   1:L PR[91] 10mm/sec FINE;
   1:  PR[GP1:91,1] = PR[GP1:90,1] + 127.618;
   1:  PR[GP1:91,2] = PR[GP1:90,2] + 91.510;
   1:L PR[91] 10mm/sec FINE;
   1:  PR[GP1:91,1] = PR[GP1:90,1] + 127.930;
   1:  PR[GP1:91,2] = PR[GP1:90,2] + 92.754;
   1:L PR[91] 10mm/sec FINE;
   1:  PR[GP1:91,1] = PR[GP1:90,1] + 128.133;
   1:  PR[GP1:91,2] = PR[GP1:90,2] + 93.973;
   1:L PR[91] 10mm/sec FINE;
   1:  PR[GP1:91,1] = PR[GP1:90,1] + 128.288;
   1:  PR[GP1:91,2] = PR[GP1:90,2] + 95.442;
   1:L PR[91] 10mm/sec FINE;
   1:  PR[GP1:91,1] = PR[GP1:90,1] + 128.356;
   1:  PR[GP1:91,2] = PR[GP1:90,2] + 96.587;
   1:L PR[91] 10mm/sec FINE;
   1:  PR[GP1:91,1] = PR[GP1:90,1] + 128.349;
   1:  PR[GP1:91,2] = PR[GP1:90,2] + 97.306;
   1:L PR[91] 10mm/sec FINE;
   1:  PR[GP1:91,1] = PR[GP1:90,1] + 128.144;
   1:  PR[GP1:91,2] = PR[GP1:90,2] + 98.735;
   1:L PR[91] 10mm/sec FINE;
   1:  PR[GP1:91,1] = PR[GP1:90,1] + 127.993;
   1:  PR[GP1:91,2] = PR[GP1:90,2] + 100.189;
   1:L PR[91] 10mm/sec FINE;
   1:  PR[GP1:91,1] = PR[GP1:90,1] + 127.642;
   1:  PR[GP1:91,2] = PR[GP1:90,2] + 101.364;
   1:L PR[91] 10mm/sec FINE;
   1:  PR[GP1:91,1] = PR[GP1:90,1] + 126.916;
   1:  PR[GP1:91,2] = PR[GP1:90,2] + 104.069;
   1:L PR[91] 10mm/sec FINE;
   1:  PR[GP1:91,1] = PR[GP1:90,1] + 125.251;
   1:  PR[GP1:91,2] = PR[GP1:90,2] + 107.811;
   1:L PR[91] 10mm/sec FINE;
   1:  PR[GP1:91,1] = PR[GP1:90,1] + 122.955;
   1:  PR[GP1:91,2] = PR[GP1:90,2] + 111.333;
   1:L PR[91] 10mm/sec FINE;
   1:  PR[GP1:91,1] = PR[GP1:90,1] + 121.825;
   1:  PR[GP1:91,2] = PR[GP1:90,2] + 112.546;
   1:L PR[91] 10mm/sec FINE;
   1:  PR[GP1:91,1] = PR[GP1:90,1] + 120.143;
   1:  PR[GP1:91,2] = PR[GP1:90,2] + 114.425;
   1:L PR[91] 10mm/sec FINE;
   1:  PR[GP1:91,1] = PR[GP1:90,1] + 118.607;
   1:  PR[GP1:91,2] = PR[GP1:90,2] + 115.642;
   1:L PR[91] 10mm/sec FINE;
   1:  PR[GP1:91,1] = PR[GP1:90,1] + 116.943;
   1:  PR[GP1:91,2] = PR[GP1:90,2] + 116.933;
   1:L PR[91] 10mm/sec FINE;
   1:  PR[GP1:91,1] = PR[GP1:90,1] + 113.463;
   1:  PR[GP1:91,2] = PR[GP1:90,2] + 118.770;
   1:L PR[91] 10mm/sec FINE;
   1:  PR[GP1:91,1] = PR[GP1:90,1] + 109.869;
   1:  PR[GP1:91,2] = PR[GP1:90,2] + 119.883;
   1:L PR[91] 10mm/sec FINE;
   1:  PR[GP1:91,1] = PR[GP1:90,1] + 108.820;
   1:  PR[GP1:91,2] = PR[GP1:90,2] + 120.007;
   1:L PR[91] 10mm/sec FINE;
   1:  PR[GP1:91,1] = PR[GP1:90,1] + 106.260;
   1:  PR[GP1:91,2] = PR[GP1:90,2] + 120.260;
   1:L PR[91] 10mm/sec FINE;
   1:  PR[GP1:91,1] = PR[GP1:90,1] + 104.599;
   1:  PR[GP1:91,2] = PR[GP1:90,2] + 120.142;
   1:L PR[91] 10mm/sec FINE;
   1:  PR[GP1:91,1] = PR[GP1:90,1] + 102.606;
   1:  PR[GP1:91,2] = PR[GP1:90,2] + 119.945;
   1:L PR[91] 10mm/sec FINE;
   1:  PR[GP1:91,1] = PR[GP1:90,1] + 101.931;
   1:  PR[GP1:91,2] = PR[GP1:90,2] + 119.914;
   1:L PR[91] 10mm/sec FINE;
   1:  PR[GP1:91,1] = PR[GP1:90,1] + 98.093;
   1:  PR[GP1:91,2] = PR[GP1:90,2] + 119.921;
   1:L PR[91] 10mm/sec FINE;
   1:  PR[GP1:91,1] = PR[GP1:90,1] + 97.212;
   1:  PR[GP1:91,2] = PR[GP1:90,2] + 119.946;
   1:L PR[91] 10mm/sec FINE;
   1:  PR[GP1:91,1] = PR[GP1:90,1] + 94.419;
   1:  PR[GP1:91,2] = PR[GP1:90,2] + 119.458;
   1:L PR[91] 10mm/sec FINE;
   1:  PR[GP1:91,1] = PR[GP1:90,1] + 92.766;
   1:  PR[GP1:91,2] = PR[GP1:90,2] + 119.217;
   1:L PR[91] 10mm/sec FINE;
   1:  PR[GP1:91,1] = PR[GP1:90,1] + 90.935;
   1:  PR[GP1:91,2] = PR[GP1:90,2] + 118.517;
   1:L PR[91] 10mm/sec FINE;
   1:  PR[GP1:91,1] = PR[GP1:90,1] + 88.767;
   1:  PR[GP1:91,2] = PR[GP1:90,2] + 117.763;
   1:L PR[91] 10mm/sec FINE;
   1:  PR[GP1:91,1] = PR[GP1:90,1] + 87.721;
   1:  PR[GP1:91,2] = PR[GP1:90,2] + 117.075;
   1:L PR[91] 10mm/sec FINE;
   1:  PR[GP1:91,1] = PR[GP1:90,1] + 85.366;
   1:  PR[GP1:91,2] = PR[GP1:90,2] + 115.642;
   1:L PR[91] 10mm/sec FINE;
   1:  PR[GP1:91,1] = PR[GP1:90,1] + 84.875;
   1:  PR[GP1:91,2] = PR[GP1:90,2] + 115.109;
   1:L PR[91] 10mm/sec FINE;
   1:  PR[GP1:91,1] = PR[GP1:90,1] + 82.710;
   1:  PR[GP1:91,2] = PR[GP1:90,2] + 112.923;
   1:L PR[91] 10mm/sec FINE;
   1:  PR[GP1:91,1] = PR[GP1:90,1] + 82.531;
   1:  PR[GP1:91,2] = PR[GP1:90,2] + 112.581;
   1:L PR[91] 10mm/sec FINE;
   1:  PR[GP1:91,1] = PR[GP1:90,1] + 80.884;
   1:  PR[GP1:91,2] = PR[GP1:90,2] + 109.710;
   1:L PR[91] 10mm/sec FINE;
   1:  PR[GP1:91,1] = PR[GP1:90,1] + 80.830;
   1:  PR[GP1:91,2] = PR[GP1:90,2] + 109.475;
   1:L PR[91] 10mm/sec FINE;
   1:  PR[GP1:91,1] = PR[GP1:90,1] + 79.909;
   1:  PR[GP1:91,2] = PR[GP1:90,2] + 106.150;
   1:L PR[91] 10mm/sec FINE;
   1:  PR[GP1:91,1] = PR[GP1:90,1] + 79.999;
   1:  PR[GP1:91,2] = PR[GP1:90,2] + 102.825;
   1:L PR[91] 10mm/sec FINE;
   1:  PR[GP1:91,1] = PR[GP1:90,1] + 80.036;
   1:  PR[GP1:91,2] = PR[GP1:90,2] + 102.315;
   1:L PR[91] 10mm/sec FINE;
   1:  PR[GP1:91,1] = PR[GP1:90,1] + 80.087;
   1:  PR[GP1:91,2] = PR[GP1:90,2] + 102.069;
   1:L PR[91] 10mm/sec FINE;
   1:  PR[GP1:91,1] = PR[GP1:90,1] + 80.782;
   1:  PR[GP1:91,2] = PR[GP1:90,2] + 99.840;
   1:L PR[91] 10mm/sec FINE;
   1:  PR[GP1:91,1] = PR[GP1:90,1] + 81.137;
   1:  PR[GP1:91,2] = PR[GP1:90,2] + 98.649;
   1:L PR[91] 10mm/sec FINE;
   1:  PR[GP1:91,1] = PR[GP1:90,1] + 81.314;
   1:  PR[GP1:91,2] = PR[GP1:90,2] + 98.024;
   1:L PR[91] 10mm/sec FINE;
   1:  PR[GP1:91,1] = PR[GP1:90,1] + 81.395;
   1:  PR[GP1:91,2] = PR[GP1:90,2] + 97.791;
   1:L PR[91] 10mm/sec FINE;
   1:  PR[GP1:91,1] = PR[GP1:90,1] + 83.374;
   1:  PR[GP1:91,2] = PR[GP1:90,2] + 94.282;
   1:L PR[91] 10mm/sec FINE;
   1:  PR[GP1:91,1] = PR[GP1:90,1] + 84.843;
   1:  PR[GP1:91,2] = PR[GP1:90,2] + 92.903;
   1:  PR[GP1:91,3] = PR[GP1:90,3] + 54.900;
   1:L PR[91] 10mm/sec FINE;
   1:  PR[GP1:91,1] = PR[GP1:90,1] + 86.776;
   1:  PR[GP1:91,2] = PR[GP1:90,2] + 90.767;
   1:L PR[91] 10mm/sec FINE;
   1:  PR[GP1:91,1] = PR[GP1:90,1] + 88.811;
   1:  PR[GP1:91,2] = PR[GP1:90,2] + 88.734;
   1:L PR[91] 10mm/sec FINE;
   1:  PR[GP1:91,1] = PR[GP1:90,1] + 90.211;
   1:  PR[GP1:91,2] = PR[GP1:90,2] + 87.682;
   1:L PR[91] 10mm/sec FINE;
   1:  PR[GP1:91,1] = PR[GP1:90,1] + 93.880;
   1:  PR[GP1:91,2] = PR[GP1:90,2] + 85.209;
   1:L PR[91] 10mm/sec FINE;
   1:  PR[GP1:91,1] = PR[GP1:90,1] + 94.184;
   1:  PR[GP1:91,2] = PR[GP1:90,2] + 85.056;
   1:L PR[91] 10mm/sec FINE;
   1:  PR[GP1:91,1] = PR[GP1:90,1] + 95.228;
   1:  PR[GP1:91,2] = PR[GP1:90,2] + 84.601;
   1:L PR[91] 10mm/sec FINE;
   1:  PR[GP1:91,1] = PR[GP1:90,1] + 99.096;
   1:  PR[GP1:91,2] = PR[GP1:90,2] + 82.673;
   1:L PR[91] 10mm/sec FINE;
   1:  PR[GP1:91,1] = PR[GP1:90,1] + 100.630;
   1:  PR[GP1:91,2] = PR[GP1:90,2] + 82.156;
   1:L PR[91] 10mm/sec FINE;
   1:  PR[GP1:91,1] = PR[GP1:90,1] + 104.317;
   1:  PR[GP1:91,2] = PR[GP1:90,2] + 81.077;
   1:L PR[91] 10mm/sec FINE;
   1:  PR[GP1:91,1] = PR[GP1:90,1] + 107.737;
   1:  PR[GP1:91,2] = PR[GP1:90,2] + 80.558;
   1:L PR[91] 10mm/sec FINE;
   1:  PR[GP1:91,1] = PR[GP1:90,1] + 109.469;
   1:  PR[GP1:91,2] = PR[GP1:90,2] + 80.392;
   1:L PR[91] 10mm/sec FINE;
   1:  PR[GP1:91,1] = PR[GP1:90,1] + 109.585;
   1:  PR[GP1:91,2] = PR[GP1:90,2] + 80.419;
   1:L PR[91] 10mm/sec FINE;
   1:  PR[GP1:91,1] = PR[GP1:90,1] + 109.851;
   1:  PR[GP1:91,2] = PR[GP1:90,2] + 80.429;
   1:L PR[91] 10mm/sec FINE;
   1:  PR[GP1:91,1] = PR[GP1:90,1] + 112.014;
   1:  PR[GP1:91,2] = PR[GP1:90,2] + 80.430;
   1:L PR[91] 10mm/sec FINE;
   1:  PR[GP1:91,1] = PR[GP1:90,1] + 113.683;
   1:  PR[GP1:91,2] = PR[GP1:90,2] + 80.515;
   1:L PR[91] 10mm/sec FINE;
   1:  PR[GP1:91,1] = PR[GP1:90,1] + 114.320;
   1:  PR[GP1:91,2] = PR[GP1:90,2] + 80.631;
   1:L PR[91] 10mm/sec FINE;
   1:  PR[GP1:91,1] = PR[GP1:90,1] + 114.818;
   1:  PR[GP1:91,2] = PR[GP1:90,2] + 80.684;
   1:L PR[91] 10mm/sec FINE;
   1:  PR[GP1:91,1] = PR[GP1:90,1] + 115.772;
   1:  PR[GP1:91,2] = PR[GP1:90,2] + 80.813;
   1:L PR[91] 10mm/sec FINE;
   1:  PR[GP1:91,1] = PR[GP1:90,1] + 117.080;
   1:  PR[GP1:91,2] = PR[GP1:90,2] + 81.097;
   1:L PR[91] 10mm/sec FINE;
   1:  PR[GP1:91,1] = PR[GP1:90,1] + 118.890;
   1:  PR[GP1:91,2] = PR[GP1:90,2] + 81.616;
   1:L PR[91] 10mm/sec FINE;
   1:  PR[GP1:91,1] = PR[GP1:90,1] + 120.940;
   1:  PR[GP1:91,2] = PR[GP1:90,2] + 82.443;
   1:L PR[91] 10mm/sec FINE;
   1:  PR[GP1:91,1] = PR[GP1:90,1] + 122.721;
   1:  PR[GP1:91,2] = PR[GP1:90,2] + 83.428;
   1:L PR[91] 10mm/sec FINE;
   1:  PR[GP1:91,1] = PR[GP1:90,1] + 123.081;
   1:  PR[GP1:91,2] = PR[GP1:90,2] + 83.673;
   1:L PR[91] 10mm/sec FINE;
   1:  PR[GP1:91,1] = PR[GP1:90,1] + 124.660;
   1:  PR[GP1:91,2] = PR[GP1:90,2] + 84.884;
   1:L PR[91] 10mm/sec FINE;
   1:  PR[GP1:91,1] = PR[GP1:90,1] + 126.251;
   1:  PR[GP1:91,2] = PR[GP1:90,2] + 86.560;
   1:L PR[91] 10mm/sec FINE;
   1:  PR[GP1:91,1] = PR[GP1:90,1] + 127.095;
   1:  PR[GP1:91,2] = PR[GP1:90,2] + 87.773;
   1:L PR[91] 10mm/sec FINE;
   1:  PR[GP1:91,1] = PR[GP1:90,1] + 127.423;
   1:  PR[GP1:91,2] = PR[GP1:90,2] + 88.315;
   1:L PR[91] 10mm/sec FINE;
   1:  PR[GP1:91,1] = PR[GP1:90,1] + 128.016;
   1:  PR[GP1:91,2] = PR[GP1:90,2] + 89.478;
   1:L PR[91] 10mm/sec FINE;
   1:  PR[GP1:91,1] = PR[GP1:90,1] + 128.433;
   1:  PR[GP1:91,2] = PR[GP1:90,2] + 90.614;
   1:L PR[91] 10mm/sec FINE;
   1:  PR[GP1:91,1] = PR[GP1:90,1] + 128.614;
   1:  PR[GP1:91,2] = PR[GP1:90,2] + 91.156;
   1:L PR[91] 10mm/sec FINE;
   1:  PR[GP1:91,1] = PR[GP1:90,1] + 128.881;
   1:  PR[GP1:91,2] = PR[GP1:90,2] + 92.221;
   1:L PR[91] 10mm/sec FINE;
   1:  PR[GP1:91,1] = PR[GP1:90,1] + 129.047;
   1:  PR[GP1:91,2] = PR[GP1:90,2] + 93.278;
   1:L PR[91] 10mm/sec FINE;
   1:  PR[GP1:91,1] = PR[GP1:90,1] + 129.087;
   1:  PR[GP1:91,2] = PR[GP1:90,2] + 93.654;
   1:L PR[91] 10mm/sec FINE;
   1:  PR[GP1:91,1] = PR[GP1:90,1] + 129.165;
   1:  PR[GP1:91,2] = PR[GP1:90,2] + 95.567;
   1:L PR[91] 10mm/sec FINE;
   1:  PR[GP1:91,1] = PR[GP1:90,1] + 129.069;
   1:  PR[GP1:91,2] = PR[GP1:90,2] + 96.744;
   1:L PR[91] 10mm/sec FINE;
   1:  PR[GP1:91,1] = PR[GP1:90,1] + 129.043;
   1:  PR[GP1:91,2] = PR[GP1:90,2] + 97.348;
   1:L PR[91] 10mm/sec FINE;
   1:  PR[GP1:91,1] = PR[GP1:90,1] + 128.780;
   1:  PR[GP1:91,2] = PR[GP1:90,2] + 99.245;
   1:L PR[91] 10mm/sec FINE;
   1:  PR[GP1:91,1] = PR[GP1:90,1] + 128.644;
   1:  PR[GP1:91,2] = PR[GP1:90,2] + 99.894;
   1:L PR[91] 10mm/sec FINE;
   1:  PR[GP1:91,1] = PR[GP1:90,1] + 128.450;
   1:  PR[GP1:91,2] = PR[GP1:90,2] + 100.521;
   1:L PR[91] 10mm/sec FINE;
   1:  PR[GP1:91,1] = PR[GP1:90,1] + 128.415;
   1:  PR[GP1:91,2] = PR[GP1:90,2] + 100.580;
   1:L PR[91] 10mm/sec FINE;
   1:  PR[GP1:91,1] = PR[GP1:90,1] + 128.092;
   1:  PR[GP1:91,2] = PR[GP1:90,2] + 101.638;
   1:L PR[91] 10mm/sec FINE;
   1:  PR[GP1:91,1] = PR[GP1:90,1] + 127.769;
   1:  PR[GP1:91,2] = PR[GP1:90,2] + 102.721;
   1:L PR[91] 10mm/sec FINE;
   1:  PR[GP1:91,1] = PR[GP1:90,1] + 127.486;
   1:  PR[GP1:91,2] = PR[GP1:90,2] + 103.770;
   1:L PR[91] 10mm/sec FINE;
   1:  PR[GP1:91,1] = PR[GP1:90,1] + 126.571;
   1:  PR[GP1:91,2] = PR[GP1:90,2] + 105.666;
   1:L PR[91] 10mm/sec FINE;
   1:  PR[GP1:91,1] = PR[GP1:90,1] + 125.764;
   1:  PR[GP1:91,2] = PR[GP1:90,2] + 107.477;
   1:L PR[91] 10mm/sec FINE;
   1:  PR[GP1:91,1] = PR[GP1:90,1] + 124.435;
   1:  PR[GP1:91,2] = PR[GP1:90,2] + 109.404;
   1:L PR[91] 10mm/sec FINE;
   1:  PR[GP1:91,1] = PR[GP1:90,1] + 123.423;
   1:  PR[GP1:91,2] = PR[GP1:90,2] + 110.957;
   1:L PR[91] 10mm/sec FINE;
   1:  PR[GP1:91,1] = PR[GP1:90,1] + 120.553;
   1:  PR[GP1:91,2] = PR[GP1:90,2] + 114.035;
   1:L PR[91] 10mm/sec FINE;
   1:  PR[GP1:91,1] = PR[GP1:90,1] + 117.335;
   1:  PR[GP1:91,2] = PR[GP1:90,2] + 116.563;
   1:L PR[91] 10mm/sec FINE;
   1:  PR[GP1:91,1] = PR[GP1:90,1] + 113.835;
   1:  PR[GP1:91,2] = PR[GP1:90,2] + 118.420;
   1:L PR[91] 10mm/sec FINE;
   1:  PR[GP1:91,1] = PR[GP1:90,1] + 110.198;
   1:  PR[GP1:91,2] = PR[GP1:90,2] + 119.557;
   1:L PR[91] 10mm/sec FINE;
   1:  PR[GP1:91,1] = PR[GP1:90,1] + 107.982;
   1:  PR[GP1:91,2] = PR[GP1:90,2] + 119.819;
   1:L PR[91] 10mm/sec FINE;
   1:  PR[GP1:91,1] = PR[GP1:90,1] + 106.531;
   1:  PR[GP1:91,2] = PR[GP1:90,2] + 119.962;
   1:L PR[91] 10mm/sec FINE;
   1:  PR[GP1:91,1] = PR[GP1:90,1] + 104.218;
   1:  PR[GP1:91,2] = PR[GP1:90,2] + 119.798;
   1:L PR[91] 10mm/sec FINE;
   1:  PR[GP1:91,1] = PR[GP1:90,1] + 103.023;
   1:  PR[GP1:91,2] = PR[GP1:90,2] + 119.685;
   1:L PR[91] 10mm/sec FINE;
   1:  PR[GP1:91,1] = PR[GP1:90,1] + 102.402;
   1:  PR[GP1:91,2] = PR[GP1:90,2] + 119.659;
   1:L PR[91] 10mm/sec FINE;
   1:  PR[GP1:91,1] = PR[GP1:90,1] + 98.454;
   1:  PR[GP1:91,2] = PR[GP1:90,2] + 119.668;
   1:L PR[91] 10mm/sec FINE;
   1:  PR[GP1:91,1] = PR[GP1:90,1] + 97.976;
   1:  PR[GP1:91,2] = PR[GP1:90,2] + 119.681;
   1:L PR[91] 10mm/sec FINE;
   1:  PR[GP1:91,1] = PR[GP1:90,1] + 94.785;
   1:  PR[GP1:91,2] = PR[GP1:90,2] + 119.124;
   1:L PR[91] 10mm/sec FINE;
   1:  PR[GP1:91,1] = PR[GP1:90,1] + 93.523;
   1:  PR[GP1:91,2] = PR[GP1:90,2] + 118.940;
   1:L PR[91] 10mm/sec FINE;
   1:  PR[GP1:91,1] = PR[GP1:90,1] + 91.321;
   1:  PR[GP1:91,2] = PR[GP1:90,2] + 118.097;
   1:L PR[91] 10mm/sec FINE;
   1:  PR[GP1:91,1] = PR[GP1:90,1] + 89.521;
   1:  PR[GP1:91,2] = PR[GP1:90,2] + 117.472;
   1:L PR[91] 10mm/sec FINE;
   1:  PR[GP1:91,1] = PR[GP1:90,1] + 88.145;
   1:  PR[GP1:91,2] = PR[GP1:90,2] + 116.567;
   1:L PR[91] 10mm/sec FINE;
   1:  PR[GP1:91,1] = PR[GP1:90,1] + 86.121;
   1:  PR[GP1:91,2] = PR[GP1:90,2] + 115.334;
   1:L PR[91] 10mm/sec FINE;
   1:  PR[GP1:91,1] = PR[GP1:90,1] + 85.359;
   1:  PR[GP1:91,2] = PR[GP1:90,2] + 114.507;
   1:L PR[91] 10mm/sec FINE;
   1:  PR[GP1:91,1] = PR[GP1:90,1] + 83.470;
   1:  PR[GP1:91,2] = PR[GP1:90,2] + 112.600;
   1:L PR[91] 10mm/sec FINE;
   1:  PR[GP1:91,1] = PR[GP1:90,1] + 83.096;
   1:  PR[GP1:91,2] = PR[GP1:90,2] + 111.886;
   1:L PR[91] 10mm/sec FINE;
   1:  PR[GP1:91,1] = PR[GP1:90,1] + 81.654;
   1:  PR[GP1:91,2] = PR[GP1:90,2] + 109.371;
   1:L PR[91] 10mm/sec FINE;
   1:  PR[GP1:91,1] = PR[GP1:90,1] + 81.497;
   1:  PR[GP1:91,2] = PR[GP1:90,2] + 108.693;
   1:L PR[91] 10mm/sec FINE;
   1:  PR[GP1:91,1] = PR[GP1:90,1] + 80.694;
   1:  PR[GP1:91,2] = PR[GP1:90,2] + 105.794;
   1:L PR[91] 10mm/sec FINE;
   1:  PR[GP1:91,1] = PR[GP1:90,1] + 80.772;
   1:  PR[GP1:91,2] = PR[GP1:90,2] + 102.897;
   1:L PR[91] 10mm/sec FINE;
   1:  PR[GP1:91,1] = PR[GP1:90,1] + 80.839;
   1:  PR[GP1:91,2] = PR[GP1:90,2] + 101.979;
   1:L PR[91] 10mm/sec FINE;
   1:  PR[GP1:91,1] = PR[GP1:90,1] + 81.532;
   1:  PR[GP1:91,2] = PR[GP1:90,2] + 99.656;
   1:L PR[91] 10mm/sec FINE;
   1:  PR[GP1:91,1] = PR[GP1:90,1] + 81.997;
   1:  PR[GP1:91,2] = PR[GP1:90,2] + 98.019;
   1:L PR[91] 10mm/sec FINE;
   1:  PR[GP1:91,1] = PR[GP1:90,1] + 82.219;
   1:  PR[GP1:91,2] = PR[GP1:90,2] + 97.376;
   1:L PR[91] 10mm/sec FINE;
   1:  PR[GP1:91,1] = PR[GP1:90,1] + 83.988;
   1:  PR[GP1:91,2] = PR[GP1:90,2] + 94.239;
   1:L PR[91] 10mm/sec FINE;
   1:  PR[GP1:91,1] = PR[GP1:90,1] + 85.706;
   1:  PR[GP1:91,2] = PR[GP1:90,2] + 92.472;
   1:  PR[GP1:91,3] = PR[GP1:90,3] + 55.900;
   1:L PR[91] 10mm/sec FINE;
   1:  PR[GP1:91,1] = PR[GP1:90,1] + 87.328;
   1:  PR[GP1:91,2] = PR[GP1:90,2] + 90.679;
   1:L PR[91] 10mm/sec FINE;
   1:  PR[GP1:91,1] = PR[GP1:90,1] + 89.714;
   1:  PR[GP1:91,2] = PR[GP1:90,2] + 88.296;
   1:L PR[91] 10mm/sec FINE;
   1:  PR[GP1:91,1] = PR[GP1:90,1] + 90.722;
   1:  PR[GP1:91,2] = PR[GP1:90,2] + 87.538;
   1:L PR[91] 10mm/sec FINE;
   1:  PR[GP1:91,1] = PR[GP1:90,1] + 94.299;
   1:  PR[GP1:91,2] = PR[GP1:90,2] + 85.127;
   1:L PR[91] 10mm/sec FINE;
   1:  PR[GP1:91,1] = PR[GP1:90,1] + 94.756;
   1:  PR[GP1:91,2] = PR[GP1:90,2] + 84.787;
   1:L PR[91] 10mm/sec FINE;
   1:  PR[GP1:91,1] = PR[GP1:90,1] + 99.777;
   1:  PR[GP1:91,2] = PR[GP1:90,2] + 82.278;
   1:L PR[91] 10mm/sec FINE;
   1:  PR[GP1:91,1] = PR[GP1:90,1] + 101.984;
   1:  PR[GP1:91,2] = PR[GP1:90,2] + 81.532;
   1:L PR[91] 10mm/sec FINE;
   1:  PR[GP1:91,1] = PR[GP1:90,1] + 104.980;
   1:  PR[GP1:91,2] = PR[GP1:90,2] + 80.656;
   1:L PR[91] 10mm/sec FINE;
   1:  PR[GP1:91,1] = PR[GP1:90,1] + 109.058;
   1:  PR[GP1:91,2] = PR[GP1:90,2] + 80.038;
   1:L PR[91] 10mm/sec FINE;
   1:  PR[GP1:91,1] = PR[GP1:90,1] + 110.125;
   1:  PR[GP1:91,2] = PR[GP1:90,2] + 79.935;
   1:L PR[91] 10mm/sec FINE;
   1:  PR[GP1:91,1] = PR[GP1:90,1] + 110.193;
   1:  PR[GP1:91,2] = PR[GP1:90,2] + 79.951;
   1:L PR[91] 10mm/sec FINE;
   1:  PR[GP1:91,1] = PR[GP1:90,1] + 110.368;
   1:  PR[GP1:91,2] = PR[GP1:90,2] + 79.957;
   1:L PR[91] 10mm/sec FINE;
   1:  PR[GP1:91,1] = PR[GP1:90,1] + 111.718;
   1:  PR[GP1:91,2] = PR[GP1:90,2] + 79.958;
   1:L PR[91] 10mm/sec FINE;
   1:  PR[GP1:91,1] = PR[GP1:90,1] + 113.477;
   1:  PR[GP1:91,2] = PR[GP1:90,2] + 80.049;
   1:L PR[91] 10mm/sec FINE;
   1:  PR[GP1:91,1] = PR[GP1:90,1] + 113.683;
   1:  PR[GP1:91,2] = PR[GP1:90,2] + 80.072;
   1:L PR[91] 10mm/sec FINE;
   1:  PR[GP1:91,1] = PR[GP1:90,1] + 115.057;
   1:  PR[GP1:91,2] = PR[GP1:90,2] + 80.057;
   1:L PR[91] 10mm/sec FINE;
   1:  PR[GP1:91,1] = PR[GP1:90,1] + 115.292;
   1:  PR[GP1:91,2] = PR[GP1:90,2] + 80.077;
   1:L PR[91] 10mm/sec FINE;
   1:  PR[GP1:91,1] = PR[GP1:90,1] + 116.479;
   1:  PR[GP1:91,2] = PR[GP1:90,2] + 80.246;
   1:L PR[91] 10mm/sec FINE;
   1:  PR[GP1:91,1] = PR[GP1:90,1] + 117.798;
   1:  PR[GP1:91,2] = PR[GP1:90,2] + 80.512;
   1:L PR[91] 10mm/sec FINE;
   1:  PR[GP1:91,1] = PR[GP1:90,1] + 118.191;
   1:  PR[GP1:91,2] = PR[GP1:90,2] + 80.607;
   1:L PR[91] 10mm/sec FINE;
   1:  PR[GP1:91,1] = PR[GP1:90,1] + 119.791;
   1:  PR[GP1:91,2] = PR[GP1:90,2] + 81.062;
   1:L PR[91] 10mm/sec FINE;
   1:  PR[GP1:91,1] = PR[GP1:90,1] + 120.343;
   1:  PR[GP1:91,2] = PR[GP1:90,2] + 81.299;
   1:L PR[91] 10mm/sec FINE;
   1:  PR[GP1:91,1] = PR[GP1:90,1] + 121.992;
   1:  PR[GP1:91,2] = PR[GP1:90,2] + 81.962;
   1:L PR[91] 10mm/sec FINE;
   1:  PR[GP1:91,1] = PR[GP1:90,1] + 123.509;
   1:  PR[GP1:91,2] = PR[GP1:90,2] + 82.800;
   1:L PR[91] 10mm/sec FINE;
   1:  PR[GP1:91,1] = PR[GP1:90,1] + 124.226;
   1:  PR[GP1:91,2] = PR[GP1:90,2] + 83.289;
   1:L PR[91] 10mm/sec FINE;
   1:  PR[GP1:91,1] = PR[GP1:90,1] + 125.545;
   1:  PR[GP1:91,2] = PR[GP1:90,2] + 84.300;
   1:L PR[91] 10mm/sec FINE;
   1:  PR[GP1:91,1] = PR[GP1:90,1] + 127.225;
   1:  PR[GP1:91,2] = PR[GP1:90,2] + 86.066;
   1:L PR[91] 10mm/sec FINE;
   1:  PR[GP1:91,1] = PR[GP1:90,1] + 127.921;
   1:  PR[GP1:91,2] = PR[GP1:90,2] + 87.066;
   1:L PR[91] 10mm/sec FINE;
   1:  PR[GP1:91,1] = PR[GP1:90,1] + 128.464;
   1:  PR[GP1:91,2] = PR[GP1:90,2] + 87.965;
   1:L PR[91] 10mm/sec FINE;
   1:  PR[GP1:91,1] = PR[GP1:90,1] + 128.952;
   1:  PR[GP1:91,2] = PR[GP1:90,2] + 88.923;
   1:L PR[91] 10mm/sec FINE;
   1:  PR[GP1:91,1] = PR[GP1:90,1] + 129.296;
   1:  PR[GP1:91,2] = PR[GP1:90,2] + 89.858;
   1:L PR[91] 10mm/sec FINE;
   1:  PR[GP1:91,1] = PR[GP1:90,1] + 129.610;
   1:  PR[GP1:91,2] = PR[GP1:90,2] + 90.804;
   1:L PR[91] 10mm/sec FINE;
   1:  PR[GP1:91,1] = PR[GP1:90,1] + 129.833;
   1:  PR[GP1:91,2] = PR[GP1:90,2] + 91.690;
   1:L PR[91] 10mm/sec FINE;
   1:  PR[GP1:91,1] = PR[GP1:90,1] + 129.970;
   1:  PR[GP1:91,2] = PR[GP1:90,2] + 92.569;
   1:L PR[91] 10mm/sec FINE;
   1:  PR[GP1:91,1] = PR[GP1:90,1] + 130.058;
   1:  PR[GP1:91,2] = PR[GP1:90,2] + 93.380;
   1:L PR[91] 10mm/sec FINE;
   1:  PR[GP1:91,1] = PR[GP1:90,1] + 130.123;
   1:  PR[GP1:91,2] = PR[GP1:90,2] + 95.001;
   1:L PR[91] 10mm/sec FINE;
   1:  PR[GP1:91,1] = PR[GP1:90,1] + 129.958;
   1:  PR[GP1:91,2] = PR[GP1:90,2] + 96.990;
   1:L PR[91] 10mm/sec FINE;
   1:  PR[GP1:91,1] = PR[GP1:90,1] + 129.717;
   1:  PR[GP1:91,2] = PR[GP1:90,2] + 98.323;
   1:L PR[91] 10mm/sec FINE;
   1:  PR[GP1:91,1] = PR[GP1:90,1] + 129.400;
   1:  PR[GP1:91,2] = PR[GP1:90,2] + 99.545;
   1:L PR[91] 10mm/sec FINE;
   1:  PR[GP1:91,1] = PR[GP1:90,1] + 129.269;
   1:  PR[GP1:91,2] = PR[GP1:90,2] + 99.979;
   1:L PR[91] 10mm/sec FINE;
   1:  PR[GP1:91,1] = PR[GP1:90,1] + 129.057;
   1:  PR[GP1:91,2] = PR[GP1:90,2] + 100.535;
   1:L PR[91] 10mm/sec FINE;
   1:  PR[GP1:91,1] = PR[GP1:90,1] + 128.701;
   1:  PR[GP1:91,2] = PR[GP1:90,2] + 101.619;
   1:L PR[91] 10mm/sec FINE;
   1:  PR[GP1:91,1] = PR[GP1:90,1] + 128.592;
   1:  PR[GP1:91,2] = PR[GP1:90,2] + 101.804;
   1:L PR[91] 10mm/sec FINE;
   1:  PR[GP1:91,1] = PR[GP1:90,1] + 128.087;
   1:  PR[GP1:91,2] = PR[GP1:90,2] + 103.462;
   1:L PR[91] 10mm/sec FINE;
   1:  PR[GP1:91,1] = PR[GP1:90,1] + 127.729;
   1:  PR[GP1:91,2] = PR[GP1:90,2] + 104.146;
   1:L PR[91] 10mm/sec FINE;
   1:  PR[GP1:91,1] = PR[GP1:90,1] + 126.284;
   1:  PR[GP1:91,2] = PR[GP1:90,2] + 107.149;
   1:L PR[91] 10mm/sec FINE;
   1:  PR[GP1:91,1] = PR[GP1:90,1] + 125.004;
   1:  PR[GP1:91,2] = PR[GP1:90,2] + 108.971;
   1:L PR[91] 10mm/sec FINE;
   1:  PR[GP1:91,1] = PR[GP1:90,1] + 123.900;
   1:  PR[GP1:91,2] = PR[GP1:90,2] + 110.588;
   1:L PR[91] 10mm/sec FINE;
   1:  PR[GP1:91,1] = PR[GP1:90,1] + 123.518;
   1:  PR[GP1:91,2] = PR[GP1:90,2] + 110.979;
   1:L PR[91] 10mm/sec FINE;
   1:  PR[GP1:91,1] = PR[GP1:90,1] + 121.012;
   1:  PR[GP1:91,2] = PR[GP1:90,2] + 113.667;
   1:L PR[91] 10mm/sec FINE;
   1:  PR[GP1:91,1] = PR[GP1:90,1] + 118.449;
   1:  PR[GP1:91,2] = PR[GP1:90,2] + 115.626;
   1:L PR[91] 10mm/sec FINE;
   1:  PR[GP1:91,1] = PR[GP1:90,1] + 117.728;
   1:  PR[GP1:91,2] = PR[GP1:90,2] + 116.194;
   1:L PR[91] 10mm/sec FINE;
   1:  PR[GP1:91,1] = PR[GP1:90,1] + 114.206;
   1:  PR[GP1:91,2] = PR[GP1:90,2] + 118.070;
   1:L PR[91] 10mm/sec FINE;
   1:  PR[GP1:91,1] = PR[GP1:90,1] + 110.528;
   1:  PR[GP1:91,2] = PR[GP1:90,2] + 119.231;
   1:L PR[91] 10mm/sec FINE;
   1:  PR[GP1:91,1] = PR[GP1:90,1] + 106.801;
   1:  PR[GP1:91,2] = PR[GP1:90,2] + 119.664;
   1:L PR[91] 10mm/sec FINE;
   1:  PR[GP1:91,1] = PR[GP1:90,1] + 103.464;
   1:  PR[GP1:91,2] = PR[GP1:90,2] + 119.419;
   1:L PR[91] 10mm/sec FINE;
   1:  PR[GP1:91,1] = PR[GP1:90,1] + 102.895;
   1:  PR[GP1:91,2] = PR[GP1:90,2] + 119.394;
   1:L PR[91] 10mm/sec FINE;
   1:  PR[GP1:91,1] = PR[GP1:90,1] + 98.742;
   1:  PR[GP1:91,2] = PR[GP1:90,2] + 119.416;
   1:L PR[91] 10mm/sec FINE;
   1:  PR[GP1:91,1] = PR[GP1:90,1] + 95.150;
   1:  PR[GP1:91,2] = PR[GP1:90,2] + 118.789;
   1:L PR[91] 10mm/sec FINE;
   1:  PR[GP1:91,1] = PR[GP1:90,1] + 94.280;
   1:  PR[GP1:91,2] = PR[GP1:90,2] + 118.662;
   1:L PR[91] 10mm/sec FINE;
   1:  PR[GP1:91,1] = PR[GP1:90,1] + 91.708;
   1:  PR[GP1:91,2] = PR[GP1:90,2] + 117.677;
   1:L PR[91] 10mm/sec FINE;
   1:  PR[GP1:91,1] = PR[GP1:90,1] + 90.276;
   1:  PR[GP1:91,2] = PR[GP1:90,2] + 117.180;
   1:L PR[91] 10mm/sec FINE;
   1:  PR[GP1:91,1] = PR[GP1:90,1] + 88.570;
   1:  PR[GP1:91,2] = PR[GP1:90,2] + 116.058;
   1:L PR[91] 10mm/sec FINE;
   1:  PR[GP1:91,1] = PR[GP1:90,1] + 86.876;
   1:  PR[GP1:91,2] = PR[GP1:90,2] + 115.027;
   1:L PR[91] 10mm/sec FINE;
   1:  PR[GP1:91,1] = PR[GP1:90,1] + 85.844;
   1:  PR[GP1:91,2] = PR[GP1:90,2] + 113.906;
   1:L PR[91] 10mm/sec FINE;
   1:  PR[GP1:91,1] = PR[GP1:90,1] + 84.230;
   1:  PR[GP1:91,2] = PR[GP1:90,2] + 112.276;
   1:L PR[91] 10mm/sec FINE;
   1:  PR[GP1:91,1] = PR[GP1:90,1] + 83.661;
   1:  PR[GP1:91,2] = PR[GP1:90,2] + 111.191;
   1:L PR[91] 10mm/sec FINE;
   1:  PR[GP1:91,1] = PR[GP1:90,1] + 82.423;
   1:  PR[GP1:91,2] = PR[GP1:90,2] + 109.032;
   1:L PR[91] 10mm/sec FINE;
   1:  PR[GP1:91,1] = PR[GP1:90,1] + 82.163;
   1:  PR[GP1:91,2] = PR[GP1:90,2] + 107.910;
   1:L PR[91] 10mm/sec FINE;
   1:  PR[GP1:91,1] = PR[GP1:90,1] + 81.479;
   1:  PR[GP1:91,2] = PR[GP1:90,2] + 105.438;
   1:L PR[91] 10mm/sec FINE;
   1:  PR[GP1:91,1] = PR[GP1:90,1] + 81.545;
   1:  PR[GP1:91,2] = PR[GP1:90,2] + 102.969;
   1:L PR[91] 10mm/sec FINE;
   1:  PR[GP1:91,1] = PR[GP1:90,1] + 81.641;
   1:  PR[GP1:91,2] = PR[GP1:90,2] + 101.620;
   1:L PR[91] 10mm/sec FINE;
   1:  PR[GP1:91,1] = PR[GP1:90,1] + 82.520;
   1:  PR[GP1:91,2] = PR[GP1:90,2] + 98.614;
   1:L PR[91] 10mm/sec FINE;
   1:  PR[GP1:91,1] = PR[GP1:90,1] + 82.680;
   1:  PR[GP1:91,2] = PR[GP1:90,2] + 98.012;
   1:L PR[91] 10mm/sec FINE;
   1:  PR[GP1:91,1] = PR[GP1:90,1] + 83.044;
   1:  PR[GP1:91,2] = PR[GP1:90,2] + 96.960;
   1:L PR[91] 10mm/sec FINE;
   1:  PR[GP1:91,1] = PR[GP1:90,1] + 84.603;
   1:  PR[GP1:91,2] = PR[GP1:90,2] + 94.196;
   1:L PR[91] 10mm/sec FINE;
   1:  PR[GP1:91,1] = PR[GP1:90,1] + 86.569;
   1:  PR[GP1:91,2] = PR[GP1:90,2] + 92.040;
   1:  PR[GP1:91,3] = PR[GP1:90,3] + 56.900;
   1:L PR[91] 10mm/sec FINE;
   1:  PR[GP1:91,1] = PR[GP1:90,1] + 87.880;
   1:  PR[GP1:91,2] = PR[GP1:90,2] + 90.590;
   1:L PR[91] 10mm/sec FINE;
   1:  PR[GP1:91,1] = PR[GP1:90,1] + 90.617;
   1:  PR[GP1:91,2] = PR[GP1:90,2] + 87.857;
   1:L PR[91] 10mm/sec FINE;
   1:  PR[GP1:91,1] = PR[GP1:90,1] + 91.233;
   1:  PR[GP1:91,2] = PR[GP1:90,2] + 87.394;
   1:L PR[91] 10mm/sec FINE;
   1:  PR[GP1:91,1] = PR[GP1:90,1] + 93.439;
   1:  PR[GP1:91,2] = PR[GP1:90,2] + 85.906;
   1:L PR[91] 10mm/sec FINE;
   1:  PR[GP1:91,1] = PR[GP1:90,1] + 95.461;
   1:  PR[GP1:91,2] = PR[GP1:90,2] + 84.405;
   1:L PR[91] 10mm/sec FINE;
   1:  PR[GP1:91,1] = PR[GP1:90,1] + 96.283;
   1:  PR[GP1:91,2] = PR[GP1:90,2] + 83.962;
   1:L PR[91] 10mm/sec FINE;
   1:  PR[GP1:91,1] = PR[GP1:90,1] + 100.457;
   1:  PR[GP1:91,2] = PR[GP1:90,2] + 81.882;
   1:L PR[91] 10mm/sec FINE;
   1:  PR[GP1:91,1] = PR[GP1:90,1] + 103.337;
   1:  PR[GP1:91,2] = PR[GP1:90,2] + 80.909;
   1:L PR[91] 10mm/sec FINE;
   1:  PR[GP1:91,1] = PR[GP1:90,1] + 105.644;
   1:  PR[GP1:91,2] = PR[GP1:90,2] + 80.234;
   1:L PR[91] 10mm/sec FINE;
   1:  PR[GP1:91,1] = PR[GP1:90,1] + 110.379;
   1:  PR[GP1:91,2] = PR[GP1:90,2] + 79.517;
   1:L PR[91] 10mm/sec FINE;
   1:  PR[GP1:91,1] = PR[GP1:90,1] + 110.804;
   1:  PR[GP1:91,2] = PR[GP1:90,2] + 79.476;
   1:L PR[91] 10mm/sec FINE;
   1:  PR[GP1:91,1] = PR[GP1:90,1] + 111.420;
   1:  PR[GP1:91,2] = PR[GP1:90,2] + 79.486;
   1:L PR[91] 10mm/sec FINE;
   1:  PR[GP1:91,1] = PR[GP1:90,1] + 112.208;
   1:  PR[GP1:91,2] = PR[GP1:90,2] + 79.532;
   1:L PR[91] 10mm/sec FINE;
   1:  PR[GP1:91,1] = PR[GP1:90,1] + 115.704;
   1:  PR[GP1:91,2] = PR[GP1:90,2] + 79.494;
   1:L PR[91] 10mm/sec FINE;
   1:  PR[GP1:91,1] = PR[GP1:90,1] + 116.329;
   1:  PR[GP1:91,2] = PR[GP1:90,2] + 79.546;
   1:L PR[91] 10mm/sec FINE;
   1:  PR[GP1:91,1] = PR[GP1:90,1] + 117.367;
   1:  PR[GP1:91,2] = PR[GP1:90,2] + 79.694;
   1:L PR[91] 10mm/sec FINE;
   1:  PR[GP1:91,1] = PR[GP1:90,1] + 118.520;
   1:  PR[GP1:91,2] = PR[GP1:90,2] + 79.927;
   1:L PR[91] 10mm/sec FINE;
   1:  PR[GP1:91,1] = PR[GP1:90,1] + 119.332;
   1:  PR[GP1:91,2] = PR[GP1:90,2] + 80.122;
   1:L PR[91] 10mm/sec FINE;
   1:  PR[GP1:91,1] = PR[GP1:90,1] + 120.694;
   1:  PR[GP1:91,2] = PR[GP1:90,2] + 80.509;
   1:L PR[91] 10mm/sec FINE;
   1:  PR[GP1:91,1] = PR[GP1:90,1] + 121.681;
   1:  PR[GP1:91,2] = PR[GP1:90,2] + 80.932;
   1:L PR[91] 10mm/sec FINE;
   1:  PR[GP1:91,1] = PR[GP1:90,1] + 123.044;
   1:  PR[GP1:91,2] = PR[GP1:90,2] + 81.480;
   1:L PR[91] 10mm/sec FINE;
   1:  PR[GP1:91,1] = PR[GP1:90,1] + 124.297;
   1:  PR[GP1:91,2] = PR[GP1:90,2] + 82.173;
   1:L PR[91] 10mm/sec FINE;
   1:  PR[GP1:91,1] = PR[GP1:90,1] + 125.370;
   1:  PR[GP1:91,2] = PR[GP1:90,2] + 82.904;
   1:L PR[91] 10mm/sec FINE;
   1:  PR[GP1:91,1] = PR[GP1:90,1] + 126.430;
   1:  PR[GP1:91,2] = PR[GP1:90,2] + 83.717;
   1:L PR[91] 10mm/sec FINE;
   1:  PR[GP1:91,1] = PR[GP1:90,1] + 128.198;
   1:  PR[GP1:91,2] = PR[GP1:90,2] + 85.572;
   1:L PR[91] 10mm/sec FINE;
   1:  PR[GP1:91,1] = PR[GP1:90,1] + 128.746;
   1:  PR[GP1:91,2] = PR[GP1:90,2] + 86.359;
   1:L PR[91] 10mm/sec FINE;
   1:  PR[GP1:91,1] = PR[GP1:90,1] + 129.505;
   1:  PR[GP1:91,2] = PR[GP1:90,2] + 87.615;
   1:L PR[91] 10mm/sec FINE;
   1:  PR[GP1:91,1] = PR[GP1:90,1] + 129.888;
   1:  PR[GP1:91,2] = PR[GP1:90,2] + 88.367;
   1:L PR[91] 10mm/sec FINE;
   1:  PR[GP1:91,1] = PR[GP1:90,1] + 130.158;
   1:  PR[GP1:91,2] = PR[GP1:90,2] + 89.102;
   1:L PR[91] 10mm/sec FINE;
   1:  PR[GP1:91,1] = PR[GP1:90,1] + 130.607;
   1:  PR[GP1:91,2] = PR[GP1:90,2] + 90.452;
   1:L PR[91] 10mm/sec FINE;
   1:  PR[GP1:91,1] = PR[GP1:90,1] + 130.785;
   1:  PR[GP1:91,2] = PR[GP1:90,2] + 91.158;
   1:L PR[91] 10mm/sec FINE;
   1:  PR[GP1:91,1] = PR[GP1:90,1] + 130.894;
   1:  PR[GP1:91,2] = PR[GP1:90,2] + 91.859;
   1:L PR[91] 10mm/sec FINE;
   1:  PR[GP1:91,1] = PR[GP1:90,1] + 131.028;
   1:  PR[GP1:91,2] = PR[GP1:90,2] + 93.106;
   1:L PR[91] 10mm/sec FINE;
   1:  PR[GP1:91,1] = PR[GP1:90,1] + 131.082;
   1:  PR[GP1:91,2] = PR[GP1:90,2] + 94.435;
   1:L PR[91] 10mm/sec FINE;
   1:  PR[GP1:91,1] = PR[GP1:90,1] + 130.895;
   1:  PR[GP1:91,2] = PR[GP1:90,2] + 96.632;
   1:L PR[91] 10mm/sec FINE;
   1:  PR[GP1:91,1] = PR[GP1:90,1] + 130.691;
   1:  PR[GP1:91,2] = PR[GP1:90,2] + 97.758;
   1:L PR[91] 10mm/sec FINE;
   1:  PR[GP1:91,1] = PR[GP1:90,1] + 130.423;
   1:  PR[GP1:91,2] = PR[GP1:90,2] + 98.792;
   1:L PR[91] 10mm/sec FINE;
   1:  PR[GP1:91,1] = PR[GP1:90,1] + 130.175;
   1:  PR[GP1:91,2] = PR[GP1:90,2] + 99.652;
   1:L PR[91] 10mm/sec FINE;
   1:  PR[GP1:91,1] = PR[GP1:90,1] + 129.205;
   1:  PR[GP1:91,2] = PR[GP1:90,2] + 102.112;
   1:L PR[91] 10mm/sec FINE;
   1:  PR[GP1:91,1] = PR[GP1:90,1] + 128.967;
   1:  PR[GP1:91,2] = PR[GP1:90,2] + 102.590;
   1:L PR[91] 10mm/sec FINE;
   1:  PR[GP1:91,1] = PR[GP1:90,1] + 128.765;
   1:  PR[GP1:91,2] = PR[GP1:90,2] + 103.041;
   1:L PR[91] 10mm/sec FINE;
   1:  PR[GP1:91,1] = PR[GP1:90,1] + 128.734;
   1:  PR[GP1:91,2] = PR[GP1:90,2] + 103.142;
   1:L PR[91] 10mm/sec FINE;
   1:  PR[GP1:91,1] = PR[GP1:90,1] + 127.349;
   1:  PR[GP1:91,2] = PR[GP1:90,2] + 105.791;
   1:L PR[91] 10mm/sec FINE;
   1:  PR[GP1:91,1] = PR[GP1:90,1] + 126.835;
   1:  PR[GP1:91,2] = PR[GP1:90,2] + 106.858;
   1:L PR[91] 10mm/sec FINE;
   1:  PR[GP1:91,1] = PR[GP1:90,1] + 126.073;
   1:  PR[GP1:91,2] = PR[GP1:90,2] + 107.877;
   1:L PR[91] 10mm/sec FINE;
   1:  PR[GP1:91,1] = PR[GP1:90,1] + 125.361;
   1:  PR[GP1:91,2] = PR[GP1:90,2] + 108.865;
   1:L PR[91] 10mm/sec FINE;
   1:  PR[GP1:91,1] = PR[GP1:90,1] + 124.397;
   1:  PR[GP1:91,2] = PR[GP1:90,2] + 110.262;
   1:L PR[91] 10mm/sec FINE;
   1:  PR[GP1:91,1] = PR[GP1:90,1] + 122.289;
   1:  PR[GP1:91,2] = PR[GP1:90,2] + 112.421;
   1:L PR[91] 10mm/sec FINE;
   1:  PR[GP1:91,1] = PR[GP1:90,1] + 121.470;
   1:  PR[GP1:91,2] = PR[GP1:90,2] + 113.299;
   1:L PR[91] 10mm/sec FINE;
   1:  PR[GP1:91,1] = PR[GP1:90,1] + 118.159;
   1:  PR[GP1:91,2] = PR[GP1:90,2] + 115.830;
   1:L PR[91] 10mm/sec FINE;
   1:  PR[GP1:91,1] = PR[GP1:90,1] + 114.579;
   1:  PR[GP1:91,2] = PR[GP1:90,2] + 117.720;
   1:L PR[91] 10mm/sec FINE;
   1:  PR[GP1:91,1] = PR[GP1:90,1] + 110.856;
   1:  PR[GP1:91,2] = PR[GP1:90,2] + 118.905;
   1:L PR[91] 10mm/sec FINE;
   1:  PR[GP1:91,1] = PR[GP1:90,1] + 107.133;
   1:  PR[GP1:91,2] = PR[GP1:90,2] + 119.347;
   1:L PR[91] 10mm/sec FINE;
   1:  PR[GP1:91,1] = PR[GP1:90,1] + 106.287;
   1:  PR[GP1:91,2] = PR[GP1:90,2] + 119.309;
   1:L PR[91] 10mm/sec FINE;
   1:  PR[GP1:91,1] = PR[GP1:90,1] + 103.935;
   1:  PR[GP1:91,2] = PR[GP1:90,2] + 119.143;
   1:L PR[91] 10mm/sec FINE;
   1:  PR[GP1:91,1] = PR[GP1:90,1] + 103.404;
   1:  PR[GP1:91,2] = PR[GP1:90,2] + 119.123;
   1:L PR[91] 10mm/sec FINE;
   1:  PR[GP1:91,1] = PR[GP1:90,1] + 100.524;
   1:  PR[GP1:91,2] = PR[GP1:90,2] + 119.134;
   1:L PR[91] 10mm/sec FINE;
   1:  PR[GP1:91,1] = PR[GP1:90,1] + 99.425;
   1:  PR[GP1:91,2] = PR[GP1:90,2] + 119.108;
   1:L PR[91] 10mm/sec FINE;
   1:  PR[GP1:91,1] = PR[GP1:90,1] + 97.820;
   1:  PR[GP1:91,2] = PR[GP1:90,2] + 118.857;
   1:L PR[91] 10mm/sec FINE;
   1:  PR[GP1:91,1] = PR[GP1:90,1] + 95.516;
   1:  PR[GP1:91,2] = PR[GP1:90,2] + 118.454;
   1:L PR[91] 10mm/sec FINE;
   1:  PR[GP1:91,1] = PR[GP1:90,1] + 95.038;
   1:  PR[GP1:91,2] = PR[GP1:90,2] + 118.384;
   1:L PR[91] 10mm/sec FINE;
   1:  PR[GP1:91,1] = PR[GP1:90,1] + 92.094;
   1:  PR[GP1:91,2] = PR[GP1:90,2] + 117.257;
   1:L PR[91] 10mm/sec FINE;
   1:  PR[GP1:91,1] = PR[GP1:90,1] + 91.030;
   1:  PR[GP1:91,2] = PR[GP1:90,2] + 116.888;
   1:L PR[91] 10mm/sec FINE;
   1:  PR[GP1:91,1] = PR[GP1:90,1] + 88.994;
   1:  PR[GP1:91,2] = PR[GP1:90,2] + 115.549;
   1:L PR[91] 10mm/sec FINE;
   1:  PR[GP1:91,1] = PR[GP1:90,1] + 87.632;
   1:  PR[GP1:91,2] = PR[GP1:90,2] + 114.720;
   1:L PR[91] 10mm/sec FINE;
   1:  PR[GP1:91,1] = PR[GP1:90,1] + 86.328;
   1:  PR[GP1:91,2] = PR[GP1:90,2] + 113.304;
   1:L PR[91] 10mm/sec FINE;
   1:  PR[GP1:91,1] = PR[GP1:90,1] + 84.990;
   1:  PR[GP1:91,2] = PR[GP1:90,2] + 111.953;
   1:L PR[91] 10mm/sec FINE;
   1:  PR[GP1:91,1] = PR[GP1:90,1] + 84.227;
   1:  PR[GP1:91,2] = PR[GP1:90,2] + 110.497;
   1:L PR[91] 10mm/sec FINE;
   1:  PR[GP1:91,1] = PR[GP1:90,1] + 83.192;
   1:  PR[GP1:91,2] = PR[GP1:90,2] + 108.693;
   1:L PR[91] 10mm/sec FINE;
   1:  PR[GP1:91,1] = PR[GP1:90,1] + 82.830;
   1:  PR[GP1:91,2] = PR[GP1:90,2] + 107.128;
   1:L PR[91] 10mm/sec FINE;
   1:  PR[GP1:91,1] = PR[GP1:90,1] + 82.264;
   1:  PR[GP1:91,2] = PR[GP1:90,2] + 105.083;
   1:L PR[91] 10mm/sec FINE;
   1:  PR[GP1:91,1] = PR[GP1:90,1] + 82.319;
   1:  PR[GP1:91,2] = PR[GP1:90,2] + 103.041;
   1:L PR[91] 10mm/sec FINE;
   1:  PR[GP1:91,1] = PR[GP1:90,1] + 82.442;
   1:  PR[GP1:91,2] = PR[GP1:90,2] + 101.253;
   1:L PR[91] 10mm/sec FINE;
   1:  PR[GP1:91,1] = PR[GP1:90,1] + 83.141;
   1:  PR[GP1:91,2] = PR[GP1:90,2] + 98.840;
   1:L PR[91] 10mm/sec FINE;
   1:  PR[GP1:91,1] = PR[GP1:90,1] + 83.362;
   1:  PR[GP1:91,2] = PR[GP1:90,2] + 98.006;
   1:L PR[91] 10mm/sec FINE;
   1:  PR[GP1:91,1] = PR[GP1:90,1] + 83.868;
   1:  PR[GP1:91,2] = PR[GP1:90,2] + 96.544;
   1:L PR[91] 10mm/sec FINE;
   1:  PR[GP1:91,1] = PR[GP1:90,1] + 85.217;
   1:  PR[GP1:91,2] = PR[GP1:90,2] + 94.152;
   1:L PR[91] 10mm/sec FINE;
   1:  PR[GP1:91,1] = PR[GP1:90,1] + 87.431;
   1:  PR[GP1:91,2] = PR[GP1:90,2] + 91.608;
   1:  PR[GP1:91,3] = PR[GP1:90,3] + 57.900;
   1:L PR[91] 10mm/sec FINE;
   1:  PR[GP1:91,1] = PR[GP1:90,1] + 88.432;
   1:  PR[GP1:91,2] = PR[GP1:90,2] + 90.502;
   1:L PR[91] 10mm/sec FINE;
   1:  PR[GP1:91,1] = PR[GP1:90,1] + 91.520;
   1:  PR[GP1:91,2] = PR[GP1:90,2] + 87.418;
   1:L PR[91] 10mm/sec FINE;
   1:  PR[GP1:91,1] = PR[GP1:90,1] + 91.744;
   1:  PR[GP1:91,2] = PR[GP1:90,2] + 87.250;
   1:L PR[91] 10mm/sec FINE;
   1:  PR[GP1:91,1] = PR[GP1:90,1] + 92.580;
   1:  PR[GP1:91,2] = PR[GP1:90,2] + 86.686;
   1:L PR[91] 10mm/sec FINE;
   1:  PR[GP1:91,1] = PR[GP1:90,1] + 96.163;
   1:  PR[GP1:91,2] = PR[GP1:90,2] + 84.024;
   1:L PR[91] 10mm/sec FINE;
   1:  PR[GP1:91,1] = PR[GP1:90,1] + 97.630;
   1:  PR[GP1:91,2] = PR[GP1:90,2] + 83.234;
   1:L PR[91] 10mm/sec FINE;
   1:  PR[GP1:91,1] = PR[GP1:90,1] + 101.137;
   1:  PR[GP1:91,2] = PR[GP1:90,2] + 81.486;
   1:L PR[91] 10mm/sec FINE;
   1:  PR[GP1:91,1] = PR[GP1:90,1] + 104.691;
   1:  PR[GP1:91,2] = PR[GP1:90,2] + 80.286;
   1:L PR[91] 10mm/sec FINE;
   1:  PR[GP1:91,1] = PR[GP1:90,1] + 106.307;
   1:  PR[GP1:91,2] = PR[GP1:90,2] + 79.813;
   1:L PR[91] 10mm/sec FINE;
   1:  PR[GP1:91,1] = PR[GP1:90,1] + 110.842;
   1:  PR[GP1:91,2] = PR[GP1:90,2] + 79.126;
   1:L PR[91] 10mm/sec FINE;
   1:  PR[GP1:91,1] = PR[GP1:90,1] + 111.519;
   1:  PR[GP1:91,2] = PR[GP1:90,2] + 78.990;
   1:L PR[91] 10mm/sec FINE;
   1:  PR[GP1:91,1] = PR[GP1:90,1] + 116.352;
   1:  PR[GP1:91,2] = PR[GP1:90,2] + 78.931;
   1:L PR[91] 10mm/sec FINE;
   1:  PR[GP1:91,1] = PR[GP1:90,1] + 117.366;
   1:  PR[GP1:91,2] = PR[GP1:90,2] + 79.015;
   1:L PR[91] 10mm/sec FINE;
   1:  PR[GP1:91,1] = PR[GP1:90,1] + 118.254;
   1:  PR[GP1:91,2] = PR[GP1:90,2] + 79.141;
   1:L PR[91] 10mm/sec FINE;
   1:  PR[GP1:91,1] = PR[GP1:90,1] + 119.243;
   1:  PR[GP1:91,2] = PR[GP1:90,2] + 79.341;
   1:L PR[91] 10mm/sec FINE;
   1:  PR[GP1:91,1] = PR[GP1:90,1] + 120.473;
   1:  PR[GP1:91,2] = PR[GP1:90,2] + 79.636;
   1:L PR[91] 10mm/sec FINE;
   1:  PR[GP1:91,1] = PR[GP1:90,1] + 121.596;
   1:  PR[GP1:91,2] = PR[GP1:90,2] + 79.956;
   1:L PR[91] 10mm/sec FINE;
   1:  PR[GP1:91,1] = PR[GP1:90,1] + 123.018;
   1:  PR[GP1:91,2] = PR[GP1:90,2] + 80.565;
   1:L PR[91] 10mm/sec FINE;
   1:  PR[GP1:91,1] = PR[GP1:90,1] + 124.096;
   1:  PR[GP1:91,2] = PR[GP1:90,2] + 80.998;
   1:L PR[91] 10mm/sec FINE;
   1:  PR[GP1:91,1] = PR[GP1:90,1] + 125.085;
   1:  PR[GP1:91,2] = PR[GP1:90,2] + 81.545;
   1:L PR[91] 10mm/sec FINE;
   1:  PR[GP1:91,1] = PR[GP1:90,1] + 126.515;
   1:  PR[GP1:91,2] = PR[GP1:90,2] + 82.520;
   1:L PR[91] 10mm/sec FINE;
   1:  PR[GP1:91,1] = PR[GP1:90,1] + 127.314;
   1:  PR[GP1:91,2] = PR[GP1:90,2] + 83.133;
   1:L PR[91] 10mm/sec FINE;
   1:  PR[GP1:91,1] = PR[GP1:90,1] + 129.172;
   1:  PR[GP1:91,2] = PR[GP1:90,2] + 85.078;
   1:L PR[91] 10mm/sec FINE;
   1:  PR[GP1:91,1] = PR[GP1:90,1] + 129.572;
   1:  PR[GP1:91,2] = PR[GP1:90,2] + 85.652;
   1:L PR[91] 10mm/sec FINE;
   1:  PR[GP1:91,1] = PR[GP1:90,1] + 130.546;
   1:  PR[GP1:91,2] = PR[GP1:90,2] + 87.265;
   1:L PR[91] 10mm/sec FINE;
   1:  PR[GP1:91,1] = PR[GP1:90,1] + 130.824;
   1:  PR[GP1:91,2] = PR[GP1:90,2] + 87.811;
   1:L PR[91] 10mm/sec FINE;
   1:  PR[GP1:91,1] = PR[GP1:90,1] + 131.021;
   1:  PR[GP1:91,2] = PR[GP1:90,2] + 88.346;
   1:L PR[91] 10mm/sec FINE;
   1:  PR[GP1:91,1] = PR[GP1:90,1] + 131.604;
   1:  PR[GP1:91,2] = PR[GP1:90,2] + 90.100;
   1:L PR[91] 10mm/sec FINE;
   1:  PR[GP1:91,1] = PR[GP1:90,1] + 131.736;
   1:  PR[GP1:91,2] = PR[GP1:90,2] + 90.626;
   1:L PR[91] 10mm/sec FINE;
   1:  PR[GP1:91,1] = PR[GP1:90,1] + 131.818;
   1:  PR[GP1:91,2] = PR[GP1:90,2] + 91.149;
   1:L PR[91] 10mm/sec FINE;
   1:  PR[GP1:91,1] = PR[GP1:90,1] + 131.999;
   1:  PR[GP1:91,2] = PR[GP1:90,2] + 92.833;
   1:L PR[91] 10mm/sec FINE;
   1:  PR[GP1:91,1] = PR[GP1:90,1] + 132.041;
   1:  PR[GP1:91,2] = PR[GP1:90,2] + 93.869;
   1:L PR[91] 10mm/sec FINE;
   1:  PR[GP1:91,1] = PR[GP1:90,1] + 131.832;
   1:  PR[GP1:91,2] = PR[GP1:90,2] + 96.274;
   1:L PR[91] 10mm/sec FINE;
   1:  PR[GP1:91,1] = PR[GP1:90,1] + 131.666;
   1:  PR[GP1:91,2] = PR[GP1:90,2] + 97.193;
   1:L PR[91] 10mm/sec FINE;
   1:  PR[GP1:91,1] = PR[GP1:90,1] + 131.447;
   1:  PR[GP1:91,2] = PR[GP1:90,2] + 98.038;
   1:L PR[91] 10mm/sec FINE;
   1:  PR[GP1:91,1] = PR[GP1:90,1] + 131.080;
   1:  PR[GP1:91,2] = PR[GP1:90,2] + 99.324;
   1:L PR[91] 10mm/sec FINE;
   1:  PR[GP1:91,1] = PR[GP1:90,1] + 130.258;
   1:  PR[GP1:91,2] = PR[GP1:90,2] + 101.413;
   1:L PR[91] 10mm/sec FINE;
   1:  PR[GP1:91,1] = PR[GP1:90,1] + 130.064;
   1:  PR[GP1:91,2] = PR[GP1:90,2] + 101.850;
   1:L PR[91] 10mm/sec FINE;
   1:  PR[GP1:91,1] = PR[GP1:90,1] + 129.398;
   1:  PR[GP1:91,2] = PR[GP1:90,2] + 103.157;
   1:L PR[91] 10mm/sec FINE;
   1:  PR[GP1:91,1] = PR[GP1:90,1] + 128.674;
   1:  PR[GP1:91,2] = PR[GP1:90,2] + 104.383;
   1:L PR[91] 10mm/sec FINE;
   1:  PR[GP1:91,1] = PR[GP1:90,1] + 128.591;
   1:  PR[GP1:91,2] = PR[GP1:90,2] + 104.321;
   1:L PR[91] 10mm/sec FINE;
   1:  PR[GP1:91,1] = PR[GP1:90,1] + 127.430;
   1:  PR[GP1:91,2] = PR[GP1:90,2] + 106.545;
   1:L PR[91] 10mm/sec FINE;
   1:  PR[GP1:91,1] = PR[GP1:90,1] + 126.835;
   1:  PR[GP1:91,2] = PR[GP1:90,2] + 107.304;
   1:L PR[91] 10mm/sec FINE;
   1:  PR[GP1:91,1] = PR[GP1:90,1] + 125.929;
   1:  PR[GP1:91,2] = PR[GP1:90,2] + 108.516;
   1:L PR[91] 10mm/sec FINE;
   1:  PR[GP1:91,1] = PR[GP1:90,1] + 124.902;
   1:  PR[GP1:91,2] = PR[GP1:90,2] + 109.942;
   1:L PR[91] 10mm/sec FINE;
   1:  PR[GP1:91,1] = PR[GP1:90,1] + 123.174;
   1:  PR[GP1:91,2] = PR[GP1:90,2] + 111.674;
   1:L PR[91] 10mm/sec FINE;
   1:  PR[GP1:91,1] = PR[GP1:90,1] + 121.942;
   1:  PR[GP1:91,2] = PR[GP1:90,2] + 112.950;
   1:L PR[91] 10mm/sec FINE;
   1:  PR[GP1:91,1] = PR[GP1:90,1] + 120.898;
   1:  PR[GP1:91,2] = PR[GP1:90,2] + 113.719;
   1:L PR[91] 10mm/sec FINE;
   1:  PR[GP1:91,1] = PR[GP1:90,1] + 118.606;
   1:  PR[GP1:91,2] = PR[GP1:90,2] + 115.470;
   1:L PR[91] 10mm/sec FINE;
   1:  PR[GP1:91,1] = PR[GP1:90,1] + 114.992;
   1:  PR[GP1:91,2] = PR[GP1:90,2] + 117.368;
   1:L PR[91] 10mm/sec FINE;
   1:  PR[GP1:91,1] = PR[GP1:90,1] + 111.245;
   1:  PR[GP1:91,2] = PR[GP1:90,2] + 118.565;
   1:L PR[91] 10mm/sec FINE;
   1:  PR[GP1:91,1] = PR[GP1:90,1] + 107.499;
   1:  PR[GP1:91,2] = PR[GP1:90,2] + 119.022;
   1:L PR[91] 10mm/sec FINE;
   1:  PR[GP1:91,1] = PR[GP1:90,1] + 106.221;
   1:  PR[GP1:91,2] = PR[GP1:90,2] + 118.976;
   1:L PR[91] 10mm/sec FINE;
   1:  PR[GP1:91,1] = PR[GP1:90,1] + 104.428;
   1:  PR[GP1:91,2] = PR[GP1:90,2] + 118.859;
   1:L PR[91] 10mm/sec FINE;
   1:  PR[GP1:91,1] = PR[GP1:90,1] + 103.946;
   1:  PR[GP1:91,2] = PR[GP1:90,2] + 118.841;
   1:L PR[91] 10mm/sec FINE;
   1:  PR[GP1:91,1] = PR[GP1:90,1] + 101.769;
   1:L PR[91] 10mm/sec FINE;
   1:  PR[GP1:91,1] = PR[GP1:90,1] + 100.083;
   1:  PR[GP1:91,2] = PR[GP1:90,2] + 118.786;
   1:L PR[91] 10mm/sec FINE;
   1:  PR[GP1:91,1] = PR[GP1:90,1] + 95.796;
   1:  PR[GP1:91,2] = PR[GP1:90,2] + 118.107;
   1:L PR[91] 10mm/sec FINE;
   1:  PR[GP1:91,1] = PR[GP1:90,1] + 92.480;
   1:  PR[GP1:91,2] = PR[GP1:90,2] + 116.838;
   1:L PR[91] 10mm/sec FINE;
   1:  PR[GP1:91,1] = PR[GP1:90,1] + 91.784;
   1:  PR[GP1:91,2] = PR[GP1:90,2] + 116.596;
   1:L PR[91] 10mm/sec FINE;
   1:  PR[GP1:91,1] = PR[GP1:90,1] + 89.419;
   1:  PR[GP1:91,2] = PR[GP1:90,2] + 115.040;
   1:L PR[91] 10mm/sec FINE;
   1:  PR[GP1:91,1] = PR[GP1:90,1] + 88.387;
   1:  PR[GP1:91,2] = PR[GP1:90,2] + 114.412;
   1:L PR[91] 10mm/sec FINE;
   1:  PR[GP1:91,1] = PR[GP1:90,1] + 86.812;
   1:  PR[GP1:91,2] = PR[GP1:90,2] + 112.703;
   1:L PR[91] 10mm/sec FINE;
   1:  PR[GP1:91,1] = PR[GP1:90,1] + 85.750;
   1:  PR[GP1:91,2] = PR[GP1:90,2] + 111.630;
   1:L PR[91] 10mm/sec FINE;
   1:  PR[GP1:91,1] = PR[GP1:90,1] + 84.792;
   1:  PR[GP1:91,2] = PR[GP1:90,2] + 109.802;
   1:L PR[91] 10mm/sec FINE;
   1:  PR[GP1:91,1] = PR[GP1:90,1] + 83.961;
   1:  PR[GP1:91,2] = PR[GP1:90,2] + 108.354;
   1:L PR[91] 10mm/sec FINE;
   1:  PR[GP1:91,1] = PR[GP1:90,1] + 83.497;
   1:  PR[GP1:91,2] = PR[GP1:90,2] + 106.345;
   1:L PR[91] 10mm/sec FINE;
   1:  PR[GP1:91,1] = PR[GP1:90,1] + 83.048;
   1:  PR[GP1:91,2] = PR[GP1:90,2] + 104.727;
   1:L PR[91] 10mm/sec FINE;
   1:  PR[GP1:91,1] = PR[GP1:90,1] + 83.092;
   1:  PR[GP1:91,2] = PR[GP1:90,2] + 103.113;
   1:L PR[91] 10mm/sec FINE;
   1:  PR[GP1:91,1] = PR[GP1:90,1] + 83.241;
   1:  PR[GP1:91,2] = PR[GP1:90,2] + 100.866;
   1:L PR[91] 10mm/sec FINE;
   1:  PR[GP1:91,1] = PR[GP1:90,1] + 83.762;
   1:  PR[GP1:91,2] = PR[GP1:90,2] + 99.067;
   1:L PR[91] 10mm/sec FINE;
   1:  PR[GP1:91,1] = PR[GP1:90,1] + 84.045;
   1:  PR[GP1:91,2] = PR[GP1:90,2] + 98.001;
   1:L PR[91] 10mm/sec FINE;
   1:  PR[GP1:91,1] = PR[GP1:90,1] + 84.692;
   1:  PR[GP1:91,2] = PR[GP1:90,2] + 96.128;
   1:L PR[91] 10mm/sec FINE;
   1:  PR[GP1:91,1] = PR[GP1:90,1] + 85.831;
   1:  PR[GP1:91,2] = PR[GP1:90,2] + 94.109;
   1:L PR[91] 10mm/sec FINE;
   1:  PR[GP1:91,1] = PR[GP1:90,1] + 88.294;
   1:  PR[GP1:91,2] = PR[GP1:90,2] + 91.176;
   1:  PR[GP1:91,3] = PR[GP1:90,3] + 58.900;
   1:L PR[91] 10mm/sec FINE;
   1:  PR[GP1:91,1] = PR[GP1:90,1] + 88.984;
   1:  PR[GP1:91,2] = PR[GP1:90,2] + 90.414;
   1:L PR[91] 10mm/sec FINE;
   1:  PR[GP1:91,1] = PR[GP1:90,1] + 91.812;
   1:  PR[GP1:91,2] = PR[GP1:90,2] + 87.589;
   1:L PR[91] 10mm/sec FINE;
   1:  PR[GP1:91,1] = PR[GP1:90,1] + 92.358;
   1:  PR[GP1:91,2] = PR[GP1:90,2] + 87.000;
   1:L PR[91] 10mm/sec FINE;
   1:  PR[GP1:91,1] = PR[GP1:90,1] + 92.565;
   1:  PR[GP1:91,2] = PR[GP1:90,2] + 86.838;
   1:L PR[91] 10mm/sec FINE;
   1:  PR[GP1:91,1] = PR[GP1:90,1] + 96.865;
   1:  PR[GP1:91,2] = PR[GP1:90,2] + 83.643;
   1:L PR[91] 10mm/sec FINE;
   1:  PR[GP1:91,1] = PR[GP1:90,1] + 98.977;
   1:  PR[GP1:91,2] = PR[GP1:90,2] + 82.506;
   1:L PR[91] 10mm/sec FINE;
   1:  PR[GP1:91,1] = PR[GP1:90,1] + 101.818;
   1:  PR[GP1:91,2] = PR[GP1:90,2] + 81.090;
   1:L PR[91] 10mm/sec FINE;
   1:  PR[GP1:91,1] = PR[GP1:90,1] + 106.045;
   1:  PR[GP1:91,2] = PR[GP1:90,2] + 79.663;
   1:L PR[91] 10mm/sec FINE;
   1:  PR[GP1:91,1] = PR[GP1:90,1] + 106.971;
   1:  PR[GP1:91,2] = PR[GP1:90,2] + 79.392;
   1:L PR[91] 10mm/sec FINE;
   1:  PR[GP1:91,1] = PR[GP1:90,1] + 109.584;
   1:  PR[GP1:91,2] = PR[GP1:90,2] + 78.996;
   1:L PR[91] 10mm/sec FINE;
   1:  PR[GP1:91,1] = PR[GP1:90,1] + 112.315;
   1:  PR[GP1:91,2] = PR[GP1:90,2] + 78.447;
   1:L PR[91] 10mm/sec FINE;
   1:  PR[GP1:91,1] = PR[GP1:90,1] + 112.939;
   1:  PR[GP1:91,2] = PR[GP1:90,2] + 78.411;
   1:L PR[91] 10mm/sec FINE;
   1:  PR[GP1:91,1] = PR[GP1:90,1] + 116.999;
   1:  PR[GP1:91,2] = PR[GP1:90,2] + 78.367;
   1:L PR[91] 10mm/sec FINE;
   1:  PR[GP1:91,1] = PR[GP1:90,1] + 118.403;
   1:  PR[GP1:91,2] = PR[GP1:90,2] + 78.483;
   1:L PR[91] 10mm/sec FINE;
   1:  PR[GP1:91,1] = PR[GP1:90,1] + 119.142;
   1:  PR[GP1:91,2] = PR[GP1:90,2] + 78.589;
   1:L PR[91] 10mm/sec FINE;
   1:  PR[GP1:91,1] = PR[GP1:90,1] + 119.965;
   1:  PR[GP1:91,2] = PR[GP1:90,2] + 78.755;
   1:L PR[91] 10mm/sec FINE;
   1:  PR[GP1:91,1] = PR[GP1:90,1] + 121.614;
   1:  PR[GP1:91,2] = PR[GP1:90,2] + 79.151;
   1:L PR[91] 10mm/sec FINE;
   1:  PR[GP1:91,1] = PR[GP1:90,1] + 122.499;
   1:  PR[GP1:91,2] = PR[GP1:90,2] + 79.403;
   1:L PR[91] 10mm/sec FINE;
   1:  PR[GP1:91,1] = PR[GP1:90,1] + 124.355;
   1:  PR[GP1:91,2] = PR[GP1:90,2] + 80.198;
   1:L PR[91] 10mm/sec FINE;
   1:  PR[GP1:91,1] = PR[GP1:90,1] + 125.148;
   1:  PR[GP1:91,2] = PR[GP1:90,2] + 80.517;
   1:L PR[91] 10mm/sec FINE;
   1:  PR[GP1:91,1] = PR[GP1:90,1] + 125.872;
   1:  PR[GP1:91,2] = PR[GP1:90,2] + 80.917;
   1:L PR[91] 10mm/sec FINE;
   1:  PR[GP1:91,1] = PR[GP1:90,1] + 127.660;
   1:  PR[GP1:91,2] = PR[GP1:90,2] + 82.135;
   1:L PR[91] 10mm/sec FINE;
   1:  PR[GP1:91,1] = PR[GP1:90,1] + 128.199;
   1:  PR[GP1:91,2] = PR[GP1:90,2] + 82.549;
   1:L PR[91] 10mm/sec FINE;
   1:  PR[GP1:91,1] = PR[GP1:90,1] + 130.146;
   1:  PR[GP1:91,2] = PR[GP1:90,2] + 84.584;
   1:L PR[91] 10mm/sec FINE;
   1:  PR[GP1:91,1] = PR[GP1:90,1] + 130.397;
   1:  PR[GP1:91,2] = PR[GP1:90,2] + 84.945;
   1:L PR[91] 10mm/sec FINE;
   1:  PR[GP1:91,1] = PR[GP1:90,1] + 131.587;
   1:  PR[GP1:91,2] = PR[GP1:90,2] + 86.915;
   1:L PR[91] 10mm/sec FINE;
   1:  PR[GP1:91,1] = PR[GP1:90,1] + 131.759;
   1:  PR[GP1:91,2] = PR[GP1:90,2] + 87.253;
   1:L PR[91] 10mm/sec FINE;
   1:  PR[GP1:91,1] = PR[GP1:90,1] + 132.601;
   1:  PR[GP1:91,2] = PR[GP1:90,2] + 89.748;
   1:L PR[91] 10mm/sec FINE;
   1:  PR[GP1:91,1] = PR[GP1:90,1] + 132.688;
   1:  PR[GP1:91,2] = PR[GP1:90,2] + 90.094;
   1:L PR[91] 10mm/sec FINE;
   1:  PR[GP1:91,1] = PR[GP1:90,1] + 132.742;
   1:  PR[GP1:91,2] = PR[GP1:90,2] + 90.440;
   1:L PR[91] 10mm/sec FINE;
   1:  PR[GP1:91,1] = PR[GP1:90,1] + 132.970;
   1:  PR[GP1:91,2] = PR[GP1:90,2] + 92.559;
   1:L PR[91] 10mm/sec FINE;
   1:  PR[GP1:91,1] = PR[GP1:90,1] + 133.000;
   1:  PR[GP1:91,2] = PR[GP1:90,2] + 93.303;
   1:L PR[91] 10mm/sec FINE;
   1:  PR[GP1:91,1] = PR[GP1:90,1] + 132.769;
   1:  PR[GP1:91,2] = PR[GP1:90,2] + 95.916;
   1:L PR[91] 10mm/sec FINE;
   1:  PR[GP1:91,1] = PR[GP1:90,1] + 132.640;
   1:  PR[GP1:91,2] = PR[GP1:90,2] + 96.627;
   1:L PR[91] 10mm/sec FINE;
   1:  PR[GP1:91,1] = PR[GP1:90,1] + 132.470;
   1:  PR[GP1:91,2] = PR[GP1:90,2] + 97.283;
   1:L PR[91] 10mm/sec FINE;
   1:  PR[GP1:91,1] = PR[GP1:90,1] + 131.985;
   1:  PR[GP1:91,2] = PR[GP1:90,2] + 98.997;
   1:L PR[91] 10mm/sec FINE;
   1:  PR[GP1:91,1] = PR[GP1:90,1] + 131.313;
   1:  PR[GP1:91,2] = PR[GP1:90,2] + 100.709;
   1:L PR[91] 10mm/sec FINE;
   1:  PR[GP1:91,1] = PR[GP1:90,1] + 130.953;
   1:  PR[GP1:91,2] = PR[GP1:90,2] + 101.520;
   1:L PR[91] 10mm/sec FINE;
   1:  PR[GP1:91,1] = PR[GP1:90,1] + 130.385;
   1:  PR[GP1:91,2] = PR[GP1:90,2] + 102.634;
   1:L PR[91] 10mm/sec FINE;
   1:  PR[GP1:91,1] = PR[GP1:90,1] + 129.317;
   1:  PR[GP1:91,2] = PR[GP1:90,2] + 104.420;
   1:L PR[91] 10mm/sec FINE;
   1:  PR[GP1:91,1] = PR[GP1:90,1] + 128.159;
   1:  PR[GP1:91,2] = PR[GP1:90,2] + 106.050;
   1:L PR[91] 10mm/sec FINE;
   1:  PR[GP1:91,1] = PR[GP1:90,1] + 128.075;
   1:  PR[GP1:91,2] = PR[GP1:90,2] + 106.211;
   1:L PR[91] 10mm/sec FINE;
   1:  PR[GP1:91,1] = PR[GP1:90,1] + 126.107;
   1:  PR[GP1:91,2] = PR[GP1:90,2] + 108.725;
   1:L PR[91] 10mm/sec FINE;
   1:  PR[GP1:91,1] = PR[GP1:90,1] + 125.429;
   1:  PR[GP1:91,2] = PR[GP1:90,2] + 109.650;
   1:L PR[91] 10mm/sec FINE;
   1:  PR[GP1:91,1] = PR[GP1:90,1] + 124.427;
   1:  PR[GP1:91,2] = PR[GP1:90,2] + 110.604;
   1:L PR[91] 10mm/sec FINE;
   1:  PR[GP1:91,1] = PR[GP1:90,1] + 123.419;
   1:  PR[GP1:91,2] = PR[GP1:90,2] + 111.603;
   1:L PR[91] 10mm/sec FINE;
   1:  PR[GP1:91,1] = PR[GP1:90,1] + 122.422;
   1:  PR[GP1:91,2] = PR[GP1:90,2] + 112.623;
   1:L PR[91] 10mm/sec FINE;
   1:  PR[GP1:91,1] = PR[GP1:90,1] + 121.127;
   1:  PR[GP1:91,2] = PR[GP1:90,2] + 113.563;
   1:L PR[91] 10mm/sec FINE;
   1:  PR[GP1:91,1] = PR[GP1:90,1] + 119.054;
   1:  PR[GP1:91,2] = PR[GP1:90,2] + 115.110;
   1:L PR[91] 10mm/sec FINE;
   1:  PR[GP1:91,1] = PR[GP1:90,1] + 115.424;
   1:  PR[GP1:91,2] = PR[GP1:90,2] + 117.015;
   1:L PR[91] 10mm/sec FINE;
   1:  PR[GP1:91,1] = PR[GP1:90,1] + 111.649;
   1:  PR[GP1:91,2] = PR[GP1:90,2] + 118.223;
   1:L PR[91] 10mm/sec FINE;
   1:  PR[GP1:91,1] = PR[GP1:90,1] + 109.632;
   1:  PR[GP1:91,2] = PR[GP1:90,2] + 118.486;
   1:L PR[91] 10mm/sec FINE;
   1:  PR[GP1:91,1] = PR[GP1:90,1] + 107.866;
   1:  PR[GP1:91,2] = PR[GP1:90,2] + 118.696;
   1:L PR[91] 10mm/sec FINE;
   1:  PR[GP1:91,1] = PR[GP1:90,1] + 106.548;
   1:  PR[GP1:91,2] = PR[GP1:90,2] + 118.657;
   1:L PR[91] 10mm/sec FINE;
   1:  PR[GP1:91,1] = PR[GP1:90,1] + 104.937;
   1:  PR[GP1:91,2] = PR[GP1:90,2] + 118.571;
   1:L PR[91] 10mm/sec FINE;
   1:  PR[GP1:91,1] = PR[GP1:90,1] + 102.689;
   1:  PR[GP1:91,2] = PR[GP1:90,2] + 118.541;
   1:L PR[91] 10mm/sec FINE;
   1:  PR[GP1:91,1] = PR[GP1:90,1] + 100.740;
   1:  PR[GP1:91,2] = PR[GP1:90,2] + 118.464;
   1:L PR[91] 10mm/sec FINE;
   1:  PR[GP1:91,1] = PR[GP1:90,1] + 96.866;
   1:  PR[GP1:91,2] = PR[GP1:90,2] + 117.858;
   1:L PR[91] 10mm/sec FINE;
   1:  PR[GP1:91,1] = PR[GP1:90,1] + 96.526;
   1:  PR[GP1:91,2] = PR[GP1:90,2] + 117.789;
   1:L PR[91] 10mm/sec FINE;
   1:  PR[GP1:91,1] = PR[GP1:90,1] + 94.805;
   1:  PR[GP1:91,2] = PR[GP1:90,2] + 117.160;
   1:L PR[91] 10mm/sec FINE;
   1:  PR[GP1:91,1] = PR[GP1:90,1] + 92.541;
   1:  PR[GP1:91,2] = PR[GP1:90,2] + 116.305;
   1:L PR[91] 10mm/sec FINE;
   1:  PR[GP1:91,1] = PR[GP1:90,1] + 89.843;
   1:  PR[GP1:91,2] = PR[GP1:90,2] + 114.532;
   1:L PR[91] 10mm/sec FINE;
   1:  PR[GP1:91,1] = PR[GP1:90,1] + 89.143;
   1:  PR[GP1:91,2] = PR[GP1:90,2] + 114.105;
   1:L PR[91] 10mm/sec FINE;
   1:  PR[GP1:91,1] = PR[GP1:90,1] + 87.297;
   1:  PR[GP1:91,2] = PR[GP1:90,2] + 112.101;
   1:L PR[91] 10mm/sec FINE;
   1:  PR[GP1:91,1] = PR[GP1:90,1] + 86.510;
   1:  PR[GP1:91,2] = PR[GP1:90,2] + 111.307;
   1:L PR[91] 10mm/sec FINE;
   1:  PR[GP1:91,1] = PR[GP1:90,1] + 85.357;
   1:  PR[GP1:91,2] = PR[GP1:90,2] + 109.107;
   1:L PR[91] 10mm/sec FINE;
   1:  PR[GP1:91,1] = PR[GP1:90,1] + 84.730;
   1:  PR[GP1:91,2] = PR[GP1:90,2] + 108.014;
   1:L PR[91] 10mm/sec FINE;
   1:  PR[GP1:91,1] = PR[GP1:90,1] + 84.163;
   1:  PR[GP1:91,2] = PR[GP1:90,2] + 105.563;
   1:L PR[91] 10mm/sec FINE;
   1:  PR[GP1:91,1] = PR[GP1:90,1] + 83.833;
   1:  PR[GP1:91,2] = PR[GP1:90,2] + 104.371;
   1:L PR[91] 10mm/sec FINE;
   1:  PR[GP1:91,1] = PR[GP1:90,1] + 83.865;
   1:  PR[GP1:91,2] = PR[GP1:90,2] + 103.186;
   1:L PR[91] 10mm/sec FINE;
   1:  PR[GP1:91,1] = PR[GP1:90,1] + 84.039;
   1:  PR[GP1:91,2] = PR[GP1:90,2] + 100.479;
   1:L PR[91] 10mm/sec FINE;
   1:  PR[GP1:91,1] = PR[GP1:90,1] + 84.383;
   1:  PR[GP1:91,2] = PR[GP1:90,2] + 99.293;
   1:L PR[91] 10mm/sec FINE;
   1:  PR[GP1:91,1] = PR[GP1:90,1] + 84.727;
   1:  PR[GP1:91,2] = PR[GP1:90,2] + 97.995;
   1:L PR[91] 10mm/sec FINE;
   1:  PR[GP1:91,1] = PR[GP1:90,1] + 85.517;
   1:  PR[GP1:91,2] = PR[GP1:90,2] + 95.713;
   1:L PR[91] 10mm/sec FINE;
   1:  PR[GP1:91,1] = PR[GP1:90,1] + 86.446;
   1:  PR[GP1:91,2] = PR[GP1:90,2] + 94.066;
   1:L PR[91] 10mm/sec FINE;
   1:  PR[GP1:91,1] = PR[GP1:90,1] + 89.157;
   1:  PR[GP1:91,2] = PR[GP1:90,2] + 90.744;
   1:  PR[GP1:91,3] = PR[GP1:90,3] + 59.900;
   1:L PR[91] 10mm/sec FINE;
   1:  PR[GP1:91,1] = PR[GP1:90,1] + 89.536;
   1:  PR[GP1:91,2] = PR[GP1:90,2] + 90.326;
   1:L PR[91] 10mm/sec FINE;
   1:  PR[GP1:91,1] = PR[GP1:90,1] + 91.114;
   1:  PR[GP1:91,2] = PR[GP1:90,2] + 88.749;
   1:L PR[91] 10mm/sec FINE;
   1:  PR[GP1:91,1] = PR[GP1:90,1] + 93.084;
   1:  PR[GP1:91,2] = PR[GP1:90,2] + 86.624;
   1:L PR[91] 10mm/sec FINE;
   1:  PR[GP1:91,1] = PR[GP1:90,1] + 93.862;
   1:  PR[GP1:91,2] = PR[GP1:90,2] + 86.016;
   1:L PR[91] 10mm/sec FINE;
   1:  PR[GP1:91,1] = PR[GP1:90,1] + 97.568;
   1:  PR[GP1:91,2] = PR[GP1:90,2] + 83.263;
   1:L PR[91] 10mm/sec FINE;
   1:  PR[GP1:91,1] = PR[GP1:90,1] + 100.325;
   1:  PR[GP1:91,2] = PR[GP1:90,2] + 81.778;
   1:L PR[91] 10mm/sec FINE;
   1:  PR[GP1:91,1] = PR[GP1:90,1] + 102.498;
   1:  PR[GP1:91,2] = PR[GP1:90,2] + 80.695;
   1:L PR[91] 10mm/sec FINE;
   1:  PR[GP1:91,1] = PR[GP1:90,1] + 107.399;
   1:  PR[GP1:91,2] = PR[GP1:90,2] + 79.040;
   1:L PR[91] 10mm/sec FINE;
   1:  PR[GP1:91,1] = PR[GP1:90,1] + 107.634;
   1:  PR[GP1:91,2] = PR[GP1:90,2] + 78.971;
   1:L PR[91] 10mm/sec FINE;
   1:  PR[GP1:91,1] = PR[GP1:90,1] + 108.327;
   1:  PR[GP1:91,2] = PR[GP1:90,2] + 78.866;
   1:L PR[91] 10mm/sec FINE;
   1:  PR[GP1:91,1] = PR[GP1:90,1] + 113.107;
   1:  PR[GP1:91,2] = PR[GP1:90,2] + 77.904;
   1:L PR[91] 10mm/sec FINE;
   1:  PR[GP1:91,1] = PR[GP1:90,1] + 114.211;
   1:  PR[GP1:91,2] = PR[GP1:90,2] + 77.841;
   1:L PR[91] 10mm/sec FINE;
   1:  PR[GP1:91,1] = PR[GP1:90,1] + 117.647;
   1:  PR[GP1:91,2] = PR[GP1:90,2] + 77.804;
   1:L PR[91] 10mm/sec FINE;
   1:  PR[GP1:91,1] = PR[GP1:90,1] + 119.440;
   1:  PR[GP1:91,2] = PR[GP1:90,2] + 77.952;
   1:L PR[91] 10mm/sec FINE;
   1:  PR[GP1:91,1] = PR[GP1:90,1] + 120.030;
   1:  PR[GP1:91,2] = PR[GP1:90,2] + 78.036;
   1:L PR[91] 10mm/sec FINE;
   1:  PR[GP1:91,1] = PR[GP1:90,1] + 120.687;
   1:  PR[GP1:91,2] = PR[GP1:90,2] + 78.169;
   1:L PR[91] 10mm/sec FINE;
   1:  PR[GP1:91,1] = PR[GP1:90,1] + 122.754;
   1:  PR[GP1:91,2] = PR[GP1:90,2] + 78.665;
   1:L PR[91] 10mm/sec FINE;
   1:  PR[GP1:91,1] = PR[GP1:90,1] + 123.401;
   1:  PR[GP1:91,2] = PR[GP1:90,2] + 78.850;
   1:L PR[91] 10mm/sec FINE;
   1:  PR[GP1:91,1] = PR[GP1:90,1] + 125.692;
   1:  PR[GP1:91,2] = PR[GP1:90,2] + 79.831;
   1:L PR[91] 10mm/sec FINE;
   1:  PR[GP1:91,1] = PR[GP1:90,1] + 126.200;
   1:  PR[GP1:91,2] = PR[GP1:90,2] + 80.035;
   1:L PR[91] 10mm/sec FINE;
   1:  PR[GP1:91,1] = PR[GP1:90,1] + 126.660;
   1:  PR[GP1:91,2] = PR[GP1:90,2] + 80.290;
   1:L PR[91] 10mm/sec FINE;
   1:  PR[GP1:91,1] = PR[GP1:90,1] + 128.804;
   1:  PR[GP1:91,2] = PR[GP1:90,2] + 81.751;
   1:L PR[91] 10mm/sec FINE;
   1:  PR[GP1:91,1] = PR[GP1:90,1] + 129.084;
   1:  PR[GP1:91,2] = PR[GP1:90,2] + 81.965;
   1:L PR[91] 10mm/sec FINE;
   1:  PR[GP1:91,1] = PR[GP1:90,1] + 131.120;
   1:  PR[GP1:91,2] = PR[GP1:90,2] + 84.091;
   1:L PR[91] 10mm/sec FINE;
   1:  PR[GP1:91,1] = PR[GP1:90,1] + 131.222;
   1:  PR[GP1:91,2] = PR[GP1:90,2] + 84.238;
   1:L PR[91] 10mm/sec FINE;
   1:  PR[GP1:91,1] = PR[GP1:90,1] + 132.628;
   1:  PR[GP1:91,2] = PR[GP1:90,2] + 86.565;
   1:L PR[91] 10mm/sec FINE;
   1:  PR[GP1:91,1] = PR[GP1:90,1] + 132.695;
   1:  PR[GP1:91,2] = PR[GP1:90,2] + 86.697;
   1:L PR[91] 10mm/sec FINE;
   1:  PR[GP1:91,1] = PR[GP1:90,1] + 133.597;
   1:  PR[GP1:91,2] = PR[GP1:90,2] + 89.396;
   1:L PR[91] 10mm/sec FINE;
   1:  PR[GP1:91,1] = PR[GP1:90,1] + 133.638;
   1:  PR[GP1:91,2] = PR[GP1:90,2] + 89.558;
   1:L PR[91] 10mm/sec FINE;
   1:  PR[GP1:91,1] = PR[GP1:90,1] + 133.940;
   1:  PR[GP1:91,2] = PR[GP1:90,2] + 92.285;
   1:L PR[91] 10mm/sec FINE;
   1:  PR[GP1:91,1] = PR[GP1:90,1] + 133.958;
   1:  PR[GP1:91,2] = PR[GP1:90,2] + 92.737;
   1:L PR[91] 10mm/sec FINE;
   1:  PR[GP1:91,1] = PR[GP1:90,1] + 133.705;
   1:  PR[GP1:91,2] = PR[GP1:90,2] + 95.558;
   1:L PR[91] 10mm/sec FINE;
   1:  PR[GP1:91,1] = PR[GP1:90,1] + 133.614;
   1:  PR[GP1:91,2] = PR[GP1:90,2] + 96.062;
   1:L PR[91] 10mm/sec FINE;
   1:  PR[GP1:91,1] = PR[GP1:90,1] + 133.493;
   1:  PR[GP1:91,2] = PR[GP1:90,2] + 96.529;
   1:L PR[91] 10mm/sec FINE;
   1:  PR[GP1:91,1] = PR[GP1:90,1] + 132.891;
   1:  PR[GP1:91,2] = PR[GP1:90,2] + 98.667;
   1:L PR[91] 10mm/sec FINE;
   1:  PR[GP1:91,1] = PR[GP1:90,1] + 132.367;
   1:  PR[GP1:91,2] = PR[GP1:90,2] + 100.006;
   1:L PR[91] 10mm/sec FINE;
   1:  PR[GP1:91,1] = PR[GP1:90,1] + 131.841;
   1:  PR[GP1:91,2] = PR[GP1:90,2] + 101.191;
   1:L PR[91] 10mm/sec FINE;
   1:  PR[GP1:91,1] = PR[GP1:90,1] + 131.372;
   1:  PR[GP1:91,2] = PR[GP1:90,2] + 102.112;
   1:L PR[91] 10mm/sec FINE;
   1:  PR[GP1:91,1] = PR[GP1:90,1] + 130.224;
   1:  PR[GP1:91,2] = PR[GP1:90,2] + 104.032;
   1:L PR[91] 10mm/sec FINE;
   1:  PR[GP1:91,1] = PR[GP1:90,1] + 128.949;
   1:  PR[GP1:91,2] = PR[GP1:90,2] + 105.812;
   1:L PR[91] 10mm/sec FINE;
   1:  PR[GP1:91,1] = PR[GP1:90,1] + 127.719;
   1:  PR[GP1:91,2] = PR[GP1:90,2] + 107.297;
   1:L PR[91] 10mm/sec FINE;
   1:  PR[GP1:91,1] = PR[GP1:90,1] + 127.639;
   1:  PR[GP1:91,2] = PR[GP1:90,2] + 107.242;
   1:L PR[91] 10mm/sec FINE;
   1:  PR[GP1:91,1] = PR[GP1:90,1] + 126.003;
   1:  PR[GP1:91,2] = PR[GP1:90,2] + 109.337;
   1:L PR[91] 10mm/sec FINE;
   1:  PR[GP1:91,1] = PR[GP1:90,1] + 125.705;
   1:  PR[GP1:91,2] = PR[GP1:90,2] + 109.624;
   1:L PR[91] 10mm/sec FINE;
   1:  PR[GP1:91,1] = PR[GP1:90,1] + 125.615;
   1:  PR[GP1:91,2] = PR[GP1:90,2] + 109.687;
   1:L PR[91] 10mm/sec FINE;
   1:  PR[GP1:91,1] = PR[GP1:90,1] + 124.133;
   1:  PR[GP1:91,2] = PR[GP1:90,2] + 111.093;
   1:L PR[91] 10mm/sec FINE;
   1:  PR[GP1:91,1] = PR[GP1:90,1] + 122.909;
   1:  PR[GP1:91,2] = PR[GP1:90,2] + 112.306;
   1:L PR[91] 10mm/sec FINE;
   1:  PR[GP1:91,1] = PR[GP1:90,1] + 120.740;
   1:  PR[GP1:91,2] = PR[GP1:90,2] + 113.865;
   1:L PR[91] 10mm/sec FINE;
   1:  PR[GP1:91,1] = PR[GP1:90,1] + 119.517;
   1:  PR[GP1:91,2] = PR[GP1:90,2] + 114.775;
   1:L PR[91] 10mm/sec FINE;
   1:  PR[GP1:91,1] = PR[GP1:90,1] + 118.683;
   1:  PR[GP1:91,2] = PR[GP1:90,2] + 115.193;
   1:L PR[91] 10mm/sec FINE;
   1:  PR[GP1:91,1] = PR[GP1:90,1] + 115.857;
   1:  PR[GP1:91,2] = PR[GP1:90,2] + 116.662;
   1:L PR[91] 10mm/sec FINE;
   1:  PR[GP1:91,1] = PR[GP1:90,1] + 112.055;
   1:  PR[GP1:91,2] = PR[GP1:90,2] + 117.879;
   1:L PR[91] 10mm/sec FINE;
   1:  PR[GP1:91,1] = PR[GP1:90,1] + 108.232;
   1:  PR[GP1:91,2] = PR[GP1:90,2] + 118.370;
   1:L PR[91] 10mm/sec FINE;
   1:  PR[GP1:91,1] = PR[GP1:90,1] + 106.415;
   1:  PR[GP1:91,2] = PR[GP1:90,2] + 118.316;
   1:L PR[91] 10mm/sec FINE;
   1:  PR[GP1:91,1] = PR[GP1:90,1] + 105.469;
   1:  PR[GP1:91,2] = PR[GP1:90,2] + 118.272;
   1:L PR[91] 10mm/sec FINE;
   1:  PR[GP1:91,1] = PR[GP1:90,1] + 103.553;
   1:  PR[GP1:91,2] = PR[GP1:90,2] + 118.232;
   1:L PR[91] 10mm/sec FINE;
   1:  PR[GP1:91,1] = PR[GP1:90,1] + 101.398;
   1:  PR[GP1:91,2] = PR[GP1:90,2] + 118.143;
   1:L PR[91] 10mm/sec FINE;
   1:  PR[GP1:91,1] = PR[GP1:90,1] + 98.075;
   1:  PR[GP1:91,2] = PR[GP1:90,2] + 117.622;
   1:L PR[91] 10mm/sec FINE;
   1:  PR[GP1:91,1] = PR[GP1:90,1] + 97.243;
   1:  PR[GP1:91,2] = PR[GP1:90,2] + 117.455;
   1:L PR[91] 10mm/sec FINE;
   1:  PR[GP1:91,1] = PR[GP1:90,1] + 93.292;
   1:  PR[GP1:91,2] = PR[GP1:90,2] + 116.009;
   1:L PR[91] 10mm/sec FINE;
   1:  PR[GP1:91,1] = PR[GP1:90,1] + 90.268;
   1:  PR[GP1:91,2] = PR[GP1:90,2] + 114.023;
   1:L PR[91] 10mm/sec FINE;
   1:  PR[GP1:91,1] = PR[GP1:90,1] + 89.898;
   1:  PR[GP1:91,2] = PR[GP1:90,2] + 113.798;
   1:L PR[91] 10mm/sec FINE;
   1:  PR[GP1:91,1] = PR[GP1:90,1] + 87.781;
   1:  PR[GP1:91,2] = PR[GP1:90,2] + 111.499;
   1:L PR[91] 10mm/sec FINE;
   1:  PR[GP1:91,1] = PR[GP1:90,1] + 87.270;
   1:  PR[GP1:91,2] = PR[GP1:90,2] + 110.984;
   1:L PR[91] 10mm/sec FINE;
   1:  PR[GP1:91,1] = PR[GP1:90,1] + 85.922;
   1:  PR[GP1:91,2] = PR[GP1:90,2] + 108.412;
   1:L PR[91] 10mm/sec FINE;
   1:  PR[GP1:91,1] = PR[GP1:90,1] + 85.499;
   1:  PR[GP1:91,2] = PR[GP1:90,2] + 107.675;
   1:L PR[91] 10mm/sec FINE;
   1:  PR[GP1:91,1] = PR[GP1:90,1] + 84.830;
   1:  PR[GP1:91,2] = PR[GP1:90,2] + 104.780;
   1:L PR[91] 10mm/sec FINE;
   1:  PR[GP1:91,1] = PR[GP1:90,1] + 84.618;
   1:  PR[GP1:91,2] = PR[GP1:90,2] + 104.016;
   1:L PR[91] 10mm/sec FINE;
   1:  PR[GP1:91,1] = PR[GP1:90,1] + 84.639;
   1:  PR[GP1:91,2] = PR[GP1:90,2] + 103.258;
   1:L PR[91] 10mm/sec FINE;
   1:  PR[GP1:91,1] = PR[GP1:90,1] + 84.838;
   1:  PR[GP1:91,2] = PR[GP1:90,2] + 100.090;
   1:L PR[91] 10mm/sec FINE;
   1:  PR[GP1:91,1] = PR[GP1:90,1] + 85.409;
   1:  PR[GP1:91,2] = PR[GP1:90,2] + 97.990;
   1:L PR[91] 10mm/sec FINE;
   1:  PR[GP1:91,1] = PR[GP1:90,1] + 86.341;
   1:  PR[GP1:91,2] = PR[GP1:90,2] + 95.297;
   1:L PR[91] 10mm/sec FINE;
   1:  PR[GP1:91,1] = PR[GP1:90,1] + 87.060;
   1:  PR[GP1:91,2] = PR[GP1:90,2] + 94.022;
   1:L PR[91] 10mm/sec FINE;
   1:  PR[GP1:91,1] = PR[GP1:90,1] + 90.018;
   1:  PR[GP1:91,2] = PR[GP1:90,2] + 90.316;
   1:  PR[GP1:91,3] = PR[GP1:90,3] + 60.900;
   1:L PR[91] 10mm/sec FINE;
   1:  PR[GP1:91,1] = PR[GP1:90,1] + 90.418;
   1:  PR[GP1:91,2] = PR[GP1:90,2] + 89.908;
   1:L PR[91] 10mm/sec FINE;
   1:  PR[GP1:91,1] = PR[GP1:90,1] + 93.471;
   1:  PR[GP1:91,2] = PR[GP1:90,2] + 86.599;
   1:L PR[91] 10mm/sec FINE;
   1:  PR[GP1:91,1] = PR[GP1:90,1] + 93.809;
   1:  PR[GP1:91,2] = PR[GP1:90,2] + 86.249;
   1:L PR[91] 10mm/sec FINE;
   1:  PR[GP1:91,1] = PR[GP1:90,1] + 95.158;
   1:  PR[GP1:91,2] = PR[GP1:90,2] + 85.194;
   1:L PR[91] 10mm/sec FINE;
   1:  PR[GP1:91,1] = PR[GP1:90,1] + 98.270;
   1:  PR[GP1:91,2] = PR[GP1:90,2] + 82.882;
   1:L PR[91] 10mm/sec FINE;
   1:  PR[GP1:91,1] = PR[GP1:90,1] + 101.672;
   1:  PR[GP1:91,2] = PR[GP1:90,2] + 81.050;
   1:L PR[91] 10mm/sec FINE;
   1:  PR[GP1:91,1] = PR[GP1:90,1] + 103.179;
   1:  PR[GP1:91,2] = PR[GP1:90,2] + 80.299;
   1:L PR[91] 10mm/sec FINE;
   1:  PR[GP1:91,1] = PR[GP1:90,1] + 107.209;
   1:  PR[GP1:91,2] = PR[GP1:90,2] + 78.938;
   1:L PR[91] 10mm/sec FINE;
   1:  PR[GP1:91,1] = PR[GP1:90,1] + 108.512;
   1:  PR[GP1:91,2] = PR[GP1:90,2] + 78.443;
   1:L PR[91] 10mm/sec FINE;
   1:  PR[GP1:91,1] = PR[GP1:90,1] + 113.898;
   1:  PR[GP1:91,2] = PR[GP1:90,2] + 77.362;
   1:L PR[91] 10mm/sec FINE;
   1:  PR[GP1:91,1] = PR[GP1:90,1] + 115.483;
   1:  PR[GP1:91,2] = PR[GP1:90,2] + 77.271;
   1:L PR[91] 10mm/sec FINE;
   1:  PR[GP1:91,1] = PR[GP1:90,1] + 118.295;
   1:  PR[GP1:91,2] = PR[GP1:90,2] + 77.240;
   1:L PR[91] 10mm/sec FINE;
   1:  PR[GP1:91,1] = PR[GP1:90,1] + 120.477;
   1:  PR[GP1:91,2] = PR[GP1:90,2] + 77.421;
   1:L PR[91] 10mm/sec FINE;
   1:  PR[GP1:91,1] = PR[GP1:90,1] + 120.918;
   1:  PR[GP1:91,2] = PR[GP1:90,2] + 77.484;
   1:L PR[91] 10mm/sec FINE;
   1:  PR[GP1:91,1] = PR[GP1:90,1] + 121.410;
   1:  PR[GP1:91,2] = PR[GP1:90,2] + 77.583;
   1:L PR[91] 10mm/sec FINE;
   1:  PR[GP1:91,1] = PR[GP1:90,1] + 123.895;
   1:  PR[GP1:91,2] = PR[GP1:90,2] + 78.180;
   1:L PR[91] 10mm/sec FINE;
   1:  PR[GP1:91,1] = PR[GP1:90,1] + 124.304;
   1:  PR[GP1:91,2] = PR[GP1:90,2] + 78.296;
   1:L PR[91] 10mm/sec FINE;
   1:  PR[GP1:91,1] = PR[GP1:90,1] + 127.250;
   1:  PR[GP1:91,2] = PR[GP1:90,2] + 79.552;
   1:L PR[91] 10mm/sec FINE;
   1:  PR[GP1:91,1] = PR[GP1:90,1] + 127.448;
   1:  PR[GP1:91,2] = PR[GP1:90,2] + 79.662;
   1:L PR[91] 10mm/sec FINE;
   1:  PR[GP1:91,1] = PR[GP1:90,1] + 129.973;
   1:  PR[GP1:91,2] = PR[GP1:90,2] + 81.386;
   1:L PR[91] 10mm/sec FINE;
   1:  PR[GP1:91,1] = PR[GP1:90,1] + 130.783;
   1:  PR[GP1:91,2] = PR[GP1:90,2] + 82.230;
   1:L PR[91] 10mm/sec FINE;
   1:  PR[GP1:91,1] = PR[GP1:90,1] + 132.034;
   1:  PR[GP1:91,2] = PR[GP1:90,2] + 83.566;
   1:L PR[91] 10mm/sec FINE;
   1:  PR[GP1:91,1] = PR[GP1:90,1] + 133.609;
   1:  PR[GP1:91,2] = PR[GP1:90,2] + 86.170;
   1:L PR[91] 10mm/sec FINE;
   1:  PR[GP1:91,1] = PR[GP1:90,1] + 134.591;
   1:  PR[GP1:91,2] = PR[GP1:90,2] + 89.038;
   1:L PR[91] 10mm/sec FINE;
   1:  PR[GP1:91,1] = PR[GP1:90,1] + 134.911;
   1:  PR[GP1:91,2] = PR[GP1:90,2] + 92.011;
   1:L PR[91] 10mm/sec FINE;
   1:  PR[GP1:91,1] = PR[GP1:90,1] + 134.917;
   1:  PR[GP1:91,2] = PR[GP1:90,2] + 92.171;
   1:L PR[91] 10mm/sec FINE;
   1:  PR[GP1:91,1] = PR[GP1:90,1] + 134.642;
   1:  PR[GP1:91,2] = PR[GP1:90,2] + 95.200;
   1:L PR[91] 10mm/sec FINE;
   1:  PR[GP1:91,1] = PR[GP1:90,1] + 134.589;
   1:  PR[GP1:91,2] = PR[GP1:90,2] + 95.496;
   1:L PR[91] 10mm/sec FINE;
   1:  PR[GP1:91,1] = PR[GP1:90,1] + 133.802;
   1:  PR[GP1:91,2] = PR[GP1:90,2] + 98.330;
   1:L PR[91] 10mm/sec FINE;
   1:  PR[GP1:91,1] = PR[GP1:90,1] + 133.421;
   1:  PR[GP1:91,2] = PR[GP1:90,2] + 99.302;
   1:L PR[91] 10mm/sec FINE;
   1:  PR[GP1:91,1] = PR[GP1:90,1] + 132.730;
   1:  PR[GP1:91,2] = PR[GP1:90,2] + 100.861;
   1:L PR[91] 10mm/sec FINE;
   1:  PR[GP1:91,1] = PR[GP1:90,1] + 132.359;
   1:  PR[GP1:91,2] = PR[GP1:90,2] + 101.590;
   1:L PR[91] 10mm/sec FINE;
   1:  PR[GP1:91,1] = PR[GP1:90,1] + 131.131;
   1:  PR[GP1:91,2] = PR[GP1:90,2] + 103.645;
   1:L PR[91] 10mm/sec FINE;
   1:  PR[GP1:91,1] = PR[GP1:90,1] + 130.235;
   1:  PR[GP1:91,2] = PR[GP1:90,2] + 104.908;
   1:L PR[91] 10mm/sec FINE;
   1:  PR[GP1:91,1] = PR[GP1:90,1] + 129.776;
   1:  PR[GP1:91,2] = PR[GP1:90,2] + 105.515;
   1:L PR[91] 10mm/sec FINE;
   1:  PR[GP1:91,1] = PR[GP1:90,1] + 128.475;
   1:  PR[GP1:91,2] = PR[GP1:90,2] + 107.069;
   1:L PR[91] 10mm/sec FINE;
   1:  PR[GP1:91,1] = PR[GP1:90,1] + 127.075;
   1:  PR[GP1:91,2] = PR[GP1:90,2] + 108.496;
   1:L PR[91] 10mm/sec FINE;
   1:  PR[GP1:91,1] = PR[GP1:90,1] + 126.981;
   1:  PR[GP1:91,2] = PR[GP1:90,2] + 108.601;
   1:L PR[91] 10mm/sec FINE;
   1:  PR[GP1:91,1] = PR[GP1:90,1] + 126.958;
   1:  PR[GP1:91,2] = PR[GP1:90,2] + 108.585;
   1:L PR[91] 10mm/sec FINE;
   1:  PR[GP1:91,1] = PR[GP1:90,1] + 126.632;
   1:  PR[GP1:91,2] = PR[GP1:90,2] + 109.001;
   1:L PR[91] 10mm/sec FINE;
   1:  PR[GP1:91,1] = PR[GP1:90,1] + 125.629;
   1:  PR[GP1:91,2] = PR[GP1:90,2] + 109.968;
   1:L PR[91] 10mm/sec FINE;
   1:  PR[GP1:91,1] = PR[GP1:90,1] + 125.337;
   1:  PR[GP1:91,2] = PR[GP1:90,2] + 110.171;
   1:L PR[91] 10mm/sec FINE;
   1:  PR[GP1:91,1] = PR[GP1:90,1] + 123.840;
   1:  PR[GP1:91,2] = PR[GP1:90,2] + 111.582;
   1:L PR[91] 10mm/sec FINE;
   1:  PR[GP1:91,1] = PR[GP1:90,1] + 123.410;
   1:  PR[GP1:91,2] = PR[GP1:90,2] + 112.008;
   1:L PR[91] 10mm/sec FINE;
   1:  PR[GP1:91,1] = PR[GP1:90,1] + 122.188;
   1:  PR[GP1:91,2] = PR[GP1:90,2] + 112.848;
   1:L PR[91] 10mm/sec FINE;
   1:  PR[GP1:91,1] = PR[GP1:90,1] + 119.981;
   1:  PR[GP1:91,2] = PR[GP1:90,2] + 114.444;
   1:L PR[91] 10mm/sec FINE;
   1:  PR[GP1:91,1] = PR[GP1:90,1] + 118.173;
   1:  PR[GP1:91,2] = PR[GP1:90,2] + 115.351;
   1:L PR[91] 10mm/sec FINE;
   1:  PR[GP1:91,1] = PR[GP1:90,1] + 116.299;
   1:  PR[GP1:91,2] = PR[GP1:90,2] + 116.318;
   1:L PR[91] 10mm/sec FINE;
   1:  PR[GP1:91,1] = PR[GP1:90,1] + 112.467;
   1:  PR[GP1:91,2] = PR[GP1:90,2] + 117.536;
   1:L PR[91] 10mm/sec FINE;
   1:  PR[GP1:91,1] = PR[GP1:90,1] + 108.618;
   1:  PR[GP1:91,2] = PR[GP1:90,2] + 118.038;
   1:L PR[91] 10mm/sec FINE;
   1:  PR[GP1:91,1] = PR[GP1:90,1] + 104.785;
   1:  PR[GP1:91,2] = PR[GP1:90,2] + 117.934;
   1:L PR[91] 10mm/sec FINE;
   1:  PR[GP1:91,1] = PR[GP1:90,1] + 102.055;
   1:  PR[GP1:91,2] = PR[GP1:90,2] + 117.821;
   1:L PR[91] 10mm/sec FINE;
   1:  PR[GP1:91,1] = PR[GP1:90,1] + 99.284;
   1:  PR[GP1:91,2] = PR[GP1:90,2] + 117.387;
   1:L PR[91] 10mm/sec FINE;
   1:  PR[GP1:91,1] = PR[GP1:90,1] + 97.959;
   1:  PR[GP1:91,2] = PR[GP1:90,2] + 117.121;
   1:L PR[91] 10mm/sec FINE;
   1:  PR[GP1:91,1] = PR[GP1:90,1] + 94.529;
   1:  PR[GP1:91,2] = PR[GP1:90,2] + 115.867;
   1:L PR[91] 10mm/sec FINE;
   1:  PR[GP1:91,1] = PR[GP1:90,1] + 94.069;
   1:  PR[GP1:91,2] = PR[GP1:90,2] + 115.686;
   1:L PR[91] 10mm/sec FINE;
   1:  PR[GP1:91,1] = PR[GP1:90,1] + 90.655;
   1:  PR[GP1:91,2] = PR[GP1:90,2] + 113.492;
   1:L PR[91] 10mm/sec FINE;
   1:  PR[GP1:91,1] = PR[GP1:90,1] + 88.265;
   1:  PR[GP1:91,2] = PR[GP1:90,2] + 110.898;
   1:L PR[91] 10mm/sec FINE;
   1:  PR[GP1:91,1] = PR[GP1:90,1] + 88.030;
   1:  PR[GP1:91,2] = PR[GP1:90,2] + 110.660;
   1:L PR[91] 10mm/sec FINE;
   1:  PR[GP1:91,1] = PR[GP1:90,1] + 86.487;
   1:  PR[GP1:91,2] = PR[GP1:90,2] + 107.717;
   1:L PR[91] 10mm/sec FINE;
   1:  PR[GP1:91,1] = PR[GP1:90,1] + 86.269;
   1:  PR[GP1:91,2] = PR[GP1:90,2] + 107.336;
   1:L PR[91] 10mm/sec FINE;
   1:  PR[GP1:91,1] = PR[GP1:90,1] + 85.497;
   1:  PR[GP1:91,2] = PR[GP1:90,2] + 103.998;
   1:L PR[91] 10mm/sec FINE;
   1:  PR[GP1:91,1] = PR[GP1:90,1] + 85.403;
   1:  PR[GP1:91,2] = PR[GP1:90,2] + 103.660;
   1:L PR[91] 10mm/sec FINE;
   1:  PR[GP1:91,1] = PR[GP1:90,1] + 85.412;
   1:  PR[GP1:91,2] = PR[GP1:90,2] + 103.330;
   1:L PR[91] 10mm/sec FINE;
   1:  PR[GP1:91,1] = PR[GP1:90,1] + 85.635;
   1:  PR[GP1:91,2] = PR[GP1:90,2] + 99.711;
   1:L PR[91] 10mm/sec FINE;
   1:  PR[GP1:91,1] = PR[GP1:90,1] + 86.092;
   1:  PR[GP1:91,2] = PR[GP1:90,2] + 97.984;
   1:L PR[91] 10mm/sec FINE;
   1:  PR[GP1:91,1] = PR[GP1:90,1] + 87.166;
   1:  PR[GP1:91,2] = PR[GP1:90,2] + 94.881;
   1:L PR[91] 10mm/sec FINE;
   1:  PR[GP1:91,1] = PR[GP1:90,1] + 87.675;
   1:  PR[GP1:91,2] = PR[GP1:90,2] + 93.979;
   1:L PR[91] 10mm/sec FINE;
   1:  PR[GP1:91,1] = PR[GP1:90,1] + 88.289;
   1:  PR[GP1:91,2] = PR[GP1:90,2] + 93.936;
   1:  PR[GP1:91,3] = PR[GP1:90,3] + 61.900;
   1:L PR[91] 10mm/sec FINE;
   1:  PR[GP1:91,1] = PR[GP1:90,1] + 89.905;
   1:  PR[GP1:91,2] = PR[GP1:90,2] + 91.409;
   1:L PR[91] 10mm/sec FINE;
   1:  PR[GP1:91,1] = PR[GP1:90,1] + 90.641;
   1:  PR[GP1:91,2] = PR[GP1:90,2] + 90.175;
   1:L PR[91] 10mm/sec FINE;
   1:  PR[GP1:91,1] = PR[GP1:90,1] + 90.989;
   1:  PR[GP1:91,2] = PR[GP1:90,2] + 89.693;
   1:L PR[91] 10mm/sec FINE;
   1:  PR[GP1:91,1] = PR[GP1:90,1] + 94.051;
   1:  PR[GP1:91,2] = PR[GP1:90,2] + 86.374;
   1:L PR[91] 10mm/sec FINE;
   1:  PR[GP1:91,1] = PR[GP1:90,1] + 94.535;
   1:  PR[GP1:91,2] = PR[GP1:90,2] + 85.873;
   1:L PR[91] 10mm/sec FINE;
   1:  PR[GP1:91,1] = PR[GP1:90,1] + 96.455;
   1:  PR[GP1:91,2] = PR[GP1:90,2] + 84.372;
   1:L PR[91] 10mm/sec FINE;
   1:  PR[GP1:91,1] = PR[GP1:90,1] + 98.973;
   1:  PR[GP1:91,2] = PR[GP1:90,2] + 82.501;
   1:L PR[91] 10mm/sec FINE;
   1:  PR[GP1:91,1] = PR[GP1:90,1] + 103.019;
   1:  PR[GP1:91,2] = PR[GP1:90,2] + 80.322;
   1:L PR[91] 10mm/sec FINE;
   1:  PR[GP1:91,1] = PR[GP1:90,1] + 103.859;
   1:  PR[GP1:91,2] = PR[GP1:90,2] + 79.903;
   1:L PR[91] 10mm/sec FINE;
   1:  PR[GP1:91,1] = PR[GP1:90,1] + 106.119;
   1:  PR[GP1:91,2] = PR[GP1:90,2] + 79.140;
   1:L PR[91] 10mm/sec FINE;
   1:  PR[GP1:91,1] = PR[GP1:90,1] + 109.494;
   1:  PR[GP1:91,2] = PR[GP1:90,2] + 77.858;
   1:L PR[91] 10mm/sec FINE;
   1:  PR[GP1:91,1] = PR[GP1:90,1] + 114.690;
   1:  PR[GP1:91,2] = PR[GP1:90,2] + 76.819;
   1:L PR[91] 10mm/sec FINE;
   1:  PR[GP1:91,1] = PR[GP1:90,1] + 116.755;
   1:  PR[GP1:91,2] = PR[GP1:90,2] + 76.700;
   1:L PR[91] 10mm/sec FINE;
   1:  PR[GP1:91,1] = PR[GP1:90,1] + 118.942;
   1:  PR[GP1:91,2] = PR[GP1:90,2] + 76.677;
   1:L PR[91] 10mm/sec FINE;
   1:  PR[GP1:91,1] = PR[GP1:90,1] + 121.511;
   1:  PR[GP1:91,2] = PR[GP1:90,2] + 76.890;
   1:L PR[91] 10mm/sec FINE;
   1:  PR[GP1:91,1] = PR[GP1:90,1] + 122.135;
   1:  PR[GP1:91,2] = PR[GP1:90,2] + 76.998;
   1:L PR[91] 10mm/sec FINE;
   1:  PR[GP1:91,1] = PR[GP1:90,1] + 125.210;
   1:  PR[GP1:91,2] = PR[GP1:90,2] + 77.745;
   1:L PR[91] 10mm/sec FINE;
   1:  PR[GP1:91,1] = PR[GP1:90,1] + 127.690;
   1:  PR[GP1:91,2] = PR[GP1:90,2] + 78.807;
   1:L PR[91] 10mm/sec FINE;
   1:  PR[GP1:91,1] = PR[GP1:90,1] + 128.245;
   1:  PR[GP1:91,2] = PR[GP1:90,2] + 79.064;
   1:L PR[91] 10mm/sec FINE;
   1:  PR[GP1:91,1] = PR[GP1:90,1] + 130.532;
   1:  PR[GP1:91,2] = PR[GP1:90,2] + 80.693;
   1:L PR[91] 10mm/sec FINE;
   1:  PR[GP1:91,1] = PR[GP1:90,1] + 130.942;
   1:  PR[GP1:91,2] = PR[GP1:90,2] + 81.015;
   1:L PR[91] 10mm/sec FINE;
   1:  PR[GP1:91,1] = PR[GP1:90,1] + 132.766;
   1:  PR[GP1:91,2] = PR[GP1:90,2] + 82.962;
   1:L PR[91] 10mm/sec FINE;
   1:  PR[GP1:91,1] = PR[GP1:90,1] + 133.119;
   1:  PR[GP1:91,2] = PR[GP1:90,2] + 83.488;
   1:L PR[91] 10mm/sec FINE;
   1:  PR[GP1:91,1] = PR[GP1:90,1] + 134.447;
   1:  PR[GP1:91,2] = PR[GP1:90,2] + 85.694;
   1:L PR[91] 10mm/sec FINE;
   1:  PR[GP1:91,1] = PR[GP1:90,1] + 135.446;
   1:  PR[GP1:91,2] = PR[GP1:90,2] + 88.621;
   1:L PR[91] 10mm/sec FINE;
   1:  PR[GP1:91,1] = PR[GP1:90,1] + 135.830;
   1:  PR[GP1:91,2] = PR[GP1:90,2] + 91.677;
   1:L PR[91] 10mm/sec FINE;
   1:  PR[GP1:91,1] = PR[GP1:90,1] + 135.744;
   1:  PR[GP1:91,2] = PR[GP1:90,2] + 93.032;
   1:L PR[91] 10mm/sec FINE;
   1:  PR[GP1:91,1] = PR[GP1:90,1] + 135.561;
   1:  PR[GP1:91,2] = PR[GP1:90,2] + 94.939;
   1:L PR[91] 10mm/sec FINE;
   1:  PR[GP1:91,1] = PR[GP1:90,1] + 134.713;
   1:  PR[GP1:91,2] = PR[GP1:90,2] + 97.993;
   1:L PR[91] 10mm/sec FINE;
   1:  PR[GP1:91,1] = PR[GP1:90,1] + 134.476;
   1:  PR[GP1:91,2] = PR[GP1:90,2] + 98.598;
   1:L PR[91] 10mm/sec FINE;
   1:  PR[GP1:91,1] = PR[GP1:90,1] + 133.619;
   1:  PR[GP1:91,2] = PR[GP1:90,2] + 100.531;
   1:L PR[91] 10mm/sec FINE;
   1:  PR[GP1:91,1] = PR[GP1:90,1] + 133.346;
   1:  PR[GP1:91,2] = PR[GP1:90,2] + 101.067;
   1:L PR[91] 10mm/sec FINE;
   1:  PR[GP1:91,1] = PR[GP1:90,1] + 132.037;
   1:  PR[GP1:91,2] = PR[GP1:90,2] + 103.257;
   1:L PR[91] 10mm/sec FINE;
   1:  PR[GP1:91,1] = PR[GP1:90,1] + 131.317;
   1:  PR[GP1:91,2] = PR[GP1:90,2] + 104.272;
   1:L PR[91] 10mm/sec FINE;
   1:  PR[GP1:91,1] = PR[GP1:90,1] + 130.602;
   1:  PR[GP1:91,2] = PR[GP1:90,2] + 105.220;
   1:L PR[91] 10mm/sec FINE;
   1:  PR[GP1:91,1] = PR[GP1:90,1] + 129.499;
   1:  PR[GP1:91,2] = PR[GP1:90,2] + 106.538;
   1:L PR[91] 10mm/sec FINE;
   1:  PR[GP1:91,1] = PR[GP1:90,1] + 129.021;
   1:  PR[GP1:91,2] = PR[GP1:90,2] + 107.049;
   1:L PR[91] 10mm/sec FINE;
   1:  PR[GP1:91,1] = PR[GP1:90,1] + 127.397;
   1:  PR[GP1:91,2] = PR[GP1:90,2] + 108.689;
   1:L PR[91] 10mm/sec FINE;
   1:  PR[GP1:91,1] = PR[GP1:90,1] + 126.478;
   1:  PR[GP1:91,2] = PR[GP1:90,2] + 109.514;
   1:L PR[91] 10mm/sec FINE;
   1:  PR[GP1:91,1] = PR[GP1:90,1] + 126.271;
   1:  PR[GP1:91,2] = PR[GP1:90,2] + 109.667;
   1:L PR[91] 10mm/sec FINE;
   1:  PR[GP1:91,1] = PR[GP1:90,1] + 126.220;
   1:  PR[GP1:91,2] = PR[GP1:90,2] + 109.722;
   1:L PR[91] 10mm/sec FINE;
   1:  PR[GP1:91,1] = PR[GP1:90,1] + 126.143;
   1:  PR[GP1:91,2] = PR[GP1:90,2] + 109.759;
   1:L PR[91] 10mm/sec FINE;
   1:  PR[GP1:91,1] = PR[GP1:90,1] + 126.007;
   1:  PR[GP1:91,2] = PR[GP1:90,2] + 109.873;
   1:L PR[91] 10mm/sec FINE;
   1:  PR[GP1:91,1] = PR[GP1:90,1] + 125.552;
   1:  PR[GP1:91,2] = PR[GP1:90,2] + 110.312;
   1:L PR[91] 10mm/sec FINE;
   1:  PR[GP1:91,1] = PR[GP1:90,1] + 125.059;
   1:  PR[GP1:91,2] = PR[GP1:90,2] + 110.655;
   1:L PR[91] 10mm/sec FINE;
   1:  PR[GP1:91,1] = PR[GP1:90,1] + 123.923;
   1:  PR[GP1:91,2] = PR[GP1:90,2] + 111.722;
   1:L PR[91] 10mm/sec FINE;
   1:  PR[GP1:91,1] = PR[GP1:90,1] + 123.694;
   1:  PR[GP1:91,2] = PR[GP1:90,2] + 111.885;
   1:L PR[91] 10mm/sec FINE;
   1:  PR[GP1:91,1] = PR[GP1:90,1] + 123.540;
   1:  PR[GP1:91,2] = PR[GP1:90,2] + 111.967;
   1:L PR[91] 10mm/sec FINE;
   1:  PR[GP1:91,1] = PR[GP1:90,1] + 121.782;
   1:  PR[GP1:91,2] = PR[GP1:90,2] + 113.173;
   1:L PR[91] 10mm/sec FINE;
   1:  PR[GP1:91,1] = PR[GP1:90,1] + 120.452;
   1:  PR[GP1:91,2] = PR[GP1:90,2] + 114.126;
   1:L PR[91] 10mm/sec FINE;
   1:  PR[GP1:91,1] = PR[GP1:90,1] + 119.110;
   1:  PR[GP1:91,2] = PR[GP1:90,2] + 114.782;
   1:L PR[91] 10mm/sec FINE;
   1:  PR[GP1:91,1] = PR[GP1:90,1] + 116.748;
   1:  PR[GP1:91,2] = PR[GP1:90,2] + 115.981;
   1:L PR[91] 10mm/sec FINE;
   1:  PR[GP1:91,1] = PR[GP1:90,1] + 112.901;
   1:  PR[GP1:91,2] = PR[GP1:90,2] + 117.192;
   1:L PR[91] 10mm/sec FINE;
   1:  PR[GP1:91,1] = PR[GP1:90,1] + 109.033;
   1:  PR[GP1:91,2] = PR[GP1:90,2] + 117.696;
   1:L PR[91] 10mm/sec FINE;
   1:  PR[GP1:91,1] = PR[GP1:90,1] + 108.441;
   1:L PR[91] 10mm/sec FINE;
   1:  PR[GP1:91,1] = PR[GP1:90,1] + 106.018;
   1:  PR[GP1:91,2] = PR[GP1:90,2] + 117.635;
   1:L PR[91] 10mm/sec FINE;
   1:  PR[GP1:91,1] = PR[GP1:90,1] + 102.712;
   1:  PR[GP1:91,2] = PR[GP1:90,2] + 117.499;
   1:L PR[91] 10mm/sec FINE;
   1:  PR[GP1:91,1] = PR[GP1:90,1] + 100.493;
   1:  PR[GP1:91,2] = PR[GP1:90,2] + 117.151;
   1:L PR[91] 10mm/sec FINE;
   1:  PR[GP1:91,1] = PR[GP1:90,1] + 98.675;
   1:  PR[GP1:91,2] = PR[GP1:90,2] + 116.787;
   1:L PR[91] 10mm/sec FINE;
   1:  PR[GP1:91,1] = PR[GP1:90,1] + 95.757;
   1:  PR[GP1:91,2] = PR[GP1:90,2] + 115.720;
   1:L PR[91] 10mm/sec FINE;
   1:  PR[GP1:91,1] = PR[GP1:90,1] + 94.833;
   1:  PR[GP1:91,2] = PR[GP1:90,2] + 115.357;
   1:L PR[91] 10mm/sec FINE;
   1:  PR[GP1:91,1] = PR[GP1:90,1] + 94.731;
   1:  PR[GP1:91,2] = PR[GP1:90,2] + 115.304;
   1:L PR[91] 10mm/sec FINE;
   1:  PR[GP1:91,1] = PR[GP1:90,1] + 91.492;
   1:  PR[GP1:91,2] = PR[GP1:90,2] + 113.221;
   1:L PR[91] 10mm/sec FINE;
   1:  PR[GP1:91,1] = PR[GP1:90,1] + 91.311;
   1:  PR[GP1:91,2] = PR[GP1:90,2] + 113.061;
   1:L PR[91] 10mm/sec FINE;
   1:  PR[GP1:91,1] = PR[GP1:90,1] + 88.809;
   1:  PR[GP1:91,2] = PR[GP1:90,2] + 110.359;
   1:L PR[91] 10mm/sec FINE;
   1:  PR[GP1:91,1] = PR[GP1:90,1] + 87.039;
   1:  PR[GP1:91,2] = PR[GP1:90,2] + 107.000;
   1:L PR[91] 10mm/sec FINE;
   1:  PR[GP1:91,1] = PR[GP1:90,1] + 86.188;
   1:  PR[GP1:91,2] = PR[GP1:90,2] + 103.317;
   1:L PR[91] 10mm/sec FINE;
   1:  PR[GP1:91,1] = PR[GP1:90,1] + 86.382;
   1:  PR[GP1:91,2] = PR[GP1:90,2] + 99.568;
   1:L PR[91] 10mm/sec FINE;
   1:  PR[GP1:91,1] = PR[GP1:90,1] + 86.428;
   1:  PR[GP1:91,2] = PR[GP1:90,2] + 99.286;
   1:L PR[91] 10mm/sec FINE;
   1:  PR[GP1:91,1] = PR[GP1:90,1] + 86.774;
   1:  PR[GP1:91,2] = PR[GP1:90,2] + 97.979;
   1:L PR[91] 10mm/sec FINE;
   1:  PR[GP1:91,1] = PR[GP1:90,1] + 87.990;
   1:  PR[GP1:91,2] = PR[GP1:90,2] + 94.465;
   1:L PR[91] 10mm/sec FINE;
   1:  PR[GP1:91,1] = PR[GP1:90,1] + 88.903;
   1:  PR[GP1:91,2] = PR[GP1:90,2] + 93.892;
   1:  PR[GP1:91,3] = PR[GP1:90,3] + 62.900;
   1:L PR[91] 10mm/sec FINE;
   1:  PR[GP1:91,1] = PR[GP1:90,1] + 89.425;
   1:  PR[GP1:91,2] = PR[GP1:90,2] + 93.077;
   1:L PR[91] 10mm/sec FINE;
   1:  PR[GP1:91,1] = PR[GP1:90,1] + 91.165;
   1:  PR[GP1:91,2] = PR[GP1:90,2] + 90.159;
   1:L PR[91] 10mm/sec FINE;
   1:  PR[GP1:91,1] = PR[GP1:90,1] + 92.002;
   1:  PR[GP1:91,2] = PR[GP1:90,2] + 88.999;
   1:L PR[91] 10mm/sec FINE;
   1:  PR[GP1:91,1] = PR[GP1:90,1] + 94.631;
   1:  PR[GP1:91,2] = PR[GP1:90,2] + 86.150;
   1:L PR[91] 10mm/sec FINE;
   1:  PR[GP1:91,1] = PR[GP1:90,1] + 95.261;
   1:  PR[GP1:91,2] = PR[GP1:90,2] + 85.497;
   1:L PR[91] 10mm/sec FINE;
   1:  PR[GP1:91,1] = PR[GP1:90,1] + 97.751;
   1:  PR[GP1:91,2] = PR[GP1:90,2] + 83.550;
   1:L PR[91] 10mm/sec FINE;
   1:  PR[GP1:91,1] = PR[GP1:90,1] + 99.675;
   1:  PR[GP1:91,2] = PR[GP1:90,2] + 82.121;
   1:L PR[91] 10mm/sec FINE;
   1:  PR[GP1:91,1] = PR[GP1:90,1] + 104.542;
   1:  PR[GP1:91,2] = PR[GP1:90,2] + 79.507;
   1:L PR[91] 10mm/sec FINE;
   1:  PR[GP1:91,1] = PR[GP1:90,1] + 105.029;
   1:  PR[GP1:91,2] = PR[GP1:90,2] + 79.342;
   1:L PR[91] 10mm/sec FINE;
   1:  PR[GP1:91,1] = PR[GP1:90,1] + 110.476;
   1:  PR[GP1:91,2] = PR[GP1:90,2] + 77.273;
   1:L PR[91] 10mm/sec FINE;
   1:  PR[GP1:91,1] = PR[GP1:90,1] + 115.481;
   1:  PR[GP1:91,2] = PR[GP1:90,2] + 76.277;
   1:L PR[91] 10mm/sec FINE;
   1:  PR[GP1:91,1] = PR[GP1:90,1] + 118.028;
   1:  PR[GP1:91,2] = PR[GP1:90,2] + 76.130;
   1:L PR[91] 10mm/sec FINE;
   1:  PR[GP1:91,1] = PR[GP1:90,1] + 119.590;
   1:  PR[GP1:91,2] = PR[GP1:90,2] + 76.114;
   1:L PR[91] 10mm/sec FINE;
   1:  PR[GP1:91,1] = PR[GP1:90,1] + 122.548;
   1:  PR[GP1:91,2] = PR[GP1:90,2] + 76.358;
   1:L PR[91] 10mm/sec FINE;
   1:  PR[GP1:91,1] = PR[GP1:90,1] + 122.857;
   1:  PR[GP1:91,2] = PR[GP1:90,2] + 76.412;
   1:L PR[91] 10mm/sec FINE;
   1:  PR[GP1:91,1] = PR[GP1:90,1] + 125.531;
   1:  PR[GP1:91,2] = PR[GP1:90,2] + 77.054;
   1:L PR[91] 10mm/sec FINE;
   1:  PR[GP1:91,1] = PR[GP1:90,1] + 126.023;
   1:  PR[GP1:91,2] = PR[GP1:90,2] + 77.185;
   1:L PR[91] 10mm/sec FINE;
   1:  PR[GP1:91,1] = PR[GP1:90,1] + 126.182;
   1:  PR[GP1:91,2] = PR[GP1:90,2] + 77.247;
   1:L PR[91] 10mm/sec FINE;
   1:  PR[GP1:91,1] = PR[GP1:90,1] + 129.065;
   1:  PR[GP1:91,2] = PR[GP1:90,2] + 78.577;
   1:L PR[91] 10mm/sec FINE;
   1:  PR[GP1:91,1] = PR[GP1:90,1] + 131.026;
   1:  PR[GP1:91,2] = PR[GP1:90,2] + 79.974;
   1:L PR[91] 10mm/sec FINE;
   1:  PR[GP1:91,1] = PR[GP1:90,1] + 131.930;
   1:  PR[GP1:91,2] = PR[GP1:90,2] + 80.685;
   1:L PR[91] 10mm/sec FINE;
   1:  PR[GP1:91,1] = PR[GP1:90,1] + 133.495;
   1:  PR[GP1:91,2] = PR[GP1:90,2] + 82.355;
   1:L PR[91] 10mm/sec FINE;
   1:  PR[GP1:91,1] = PR[GP1:90,1] + 134.147;
   1:  PR[GP1:91,2] = PR[GP1:90,2] + 83.326;
   1:L PR[91] 10mm/sec FINE;
   1:  PR[GP1:91,1] = PR[GP1:90,1] + 135.286;
   1:  PR[GP1:91,2] = PR[GP1:90,2] + 85.218;
   1:L PR[91] 10mm/sec FINE;
   1:  PR[GP1:91,1] = PR[GP1:90,1] + 136.033;
   1:  PR[GP1:91,2] = PR[GP1:90,2] + 87.390;
   1:L PR[91] 10mm/sec FINE;
   1:  PR[GP1:91,1] = PR[GP1:90,1] + 136.298;
   1:  PR[GP1:91,2] = PR[GP1:90,2] + 88.207;
   1:L PR[91] 10mm/sec FINE;
   1:  PR[GP1:91,1] = PR[GP1:90,1] + 136.617;
   1:  PR[GP1:91,2] = PR[GP1:90,2] + 90.707;
   1:L PR[91] 10mm/sec FINE;
   1:  PR[GP1:91,1] = PR[GP1:90,1] + 136.671;
   1:  PR[GP1:91,2] = PR[GP1:90,2] + 91.267;
   1:L PR[91] 10mm/sec FINE;
   1:  PR[GP1:91,1] = PR[GP1:90,1] + 136.464;
   1:  PR[GP1:91,2] = PR[GP1:90,2] + 94.448;
   1:L PR[91] 10mm/sec FINE;
   1:  PR[GP1:91,1] = PR[GP1:90,1] + 136.141;
   1:  PR[GP1:91,2] = PR[GP1:90,2] + 95.791;
   1:L PR[91] 10mm/sec FINE;
   1:  PR[GP1:91,1] = PR[GP1:90,1] + 135.624;
   1:  PR[GP1:91,2] = PR[GP1:90,2] + 97.655;
   1:L PR[91] 10mm/sec FINE;
   1:  PR[GP1:91,1] = PR[GP1:90,1] + 135.530;
   1:  PR[GP1:91,2] = PR[GP1:90,2] + 97.895;
   1:L PR[91] 10mm/sec FINE;
   1:  PR[GP1:91,1] = PR[GP1:90,1] + 134.507;
   1:  PR[GP1:91,2] = PR[GP1:90,2] + 100.201;
   1:L PR[91] 10mm/sec FINE;
   1:  PR[GP1:91,1] = PR[GP1:90,1] + 134.332;
   1:  PR[GP1:91,2] = PR[GP1:90,2] + 100.545;
   1:L PR[91] 10mm/sec FINE;
   1:  PR[GP1:91,1] = PR[GP1:90,1] + 132.944;
   1:  PR[GP1:91,2] = PR[GP1:90,2] + 102.870;
   1:L PR[91] 10mm/sec FINE;
   1:  PR[GP1:91,1] = PR[GP1:90,1] + 132.400;
   1:  PR[GP1:91,2] = PR[GP1:90,2] + 103.637;
   1:L PR[91] 10mm/sec FINE;
   1:  PR[GP1:91,1] = PR[GP1:90,1] + 131.427;
   1:  PR[GP1:91,2] = PR[GP1:90,2] + 104.924;
   1:L PR[91] 10mm/sec FINE;
   1:  PR[GP1:91,1] = PR[GP1:90,1] + 130.524;
   1:  PR[GP1:91,2] = PR[GP1:90,2] + 106.004;
   1:L PR[91] 10mm/sec FINE;
   1:  PR[GP1:91,1] = PR[GP1:90,1] + 129.775;
   1:  PR[GP1:91,2] = PR[GP1:90,2] + 106.807;
   1:L PR[91] 10mm/sec FINE;
   1:  PR[GP1:91,1] = PR[GP1:90,1] + 128.381;
   1:  PR[GP1:91,2] = PR[GP1:90,2] + 108.214;
   1:L PR[91] 10mm/sec FINE;
   1:  PR[GP1:91,1] = PR[GP1:90,1] + 127.225;
   1:  PR[GP1:91,2] = PR[GP1:90,2] + 109.245;
   1:L PR[91] 10mm/sec FINE;
   1:  PR[GP1:91,1] = PR[GP1:90,1] + 125.501;
   1:  PR[GP1:91,2] = PR[GP1:90,2] + 110.524;
   1:L PR[91] 10mm/sec FINE;
   1:  PR[GP1:91,1] = PR[GP1:90,1] + 125.387;
   1:  PR[GP1:91,2] = PR[GP1:90,2] + 110.689;
   1:L PR[91] 10mm/sec FINE;
   1:  PR[GP1:91,1] = PR[GP1:90,1] + 125.293;
   1:  PR[GP1:91,2] = PR[GP1:90,2] + 110.751;
   1:L PR[91] 10mm/sec FINE;
   1:  PR[GP1:91,1] = PR[GP1:90,1] + 125.079;
   1:  PR[GP1:91,2] = PR[GP1:90,2] + 110.931;
   1:L PR[91] 10mm/sec FINE;
   1:  PR[GP1:91,1] = PR[GP1:90,1] + 124.780;
   1:  PR[GP1:91,2] = PR[GP1:90,2] + 111.139;
   1:L PR[91] 10mm/sec FINE;
   1:  PR[GP1:91,1] = PR[GP1:90,1] + 124.452;
   1:  PR[GP1:91,2] = PR[GP1:90,2] + 111.447;
   1:L PR[91] 10mm/sec FINE;
   1:  PR[GP1:91,1] = PR[GP1:90,1] + 123.657;
   1:  PR[GP1:91,2] = PR[GP1:90,2] + 112.012;
   1:L PR[91] 10mm/sec FINE;
   1:  PR[GP1:91,1] = PR[GP1:90,1] + 123.152;
   1:  PR[GP1:91,2] = PR[GP1:90,2] + 112.283;
   1:L PR[91] 10mm/sec FINE;
   1:  PR[GP1:91,1] = PR[GP1:90,1] + 120.930;
   1:  PR[GP1:91,2] = PR[GP1:90,2] + 113.818;
   1:L PR[91] 10mm/sec FINE;
   1:  PR[GP1:91,1] = PR[GP1:90,1] + 119.371;
   1:  PR[GP1:91,2] = PR[GP1:90,2] + 114.559;
   1:L PR[91] 10mm/sec FINE;
   1:  PR[GP1:91,1] = PR[GP1:90,1] + 117.197;
   1:  PR[GP1:91,2] = PR[GP1:90,2] + 115.644;
   1:L PR[91] 10mm/sec FINE;
   1:  PR[GP1:91,1] = PR[GP1:90,1] + 113.335;
   1:  PR[GP1:91,2] = PR[GP1:90,2] + 116.848;
   1:L PR[91] 10mm/sec FINE;
   1:  PR[GP1:91,1] = PR[GP1:90,1] + 109.450;
   1:  PR[GP1:91,2] = PR[GP1:90,2] + 117.354;
   1:L PR[91] 10mm/sec FINE;
   1:  PR[GP1:91,1] = PR[GP1:90,1] + 108.419;
   1:L PR[91] 10mm/sec FINE;
   1:  PR[GP1:91,1] = PR[GP1:90,1] + 107.129;
   1:  PR[GP1:91,2] = PR[GP1:90,2] + 117.331;
   1:L PR[91] 10mm/sec FINE;
   1:  PR[GP1:91,1] = PR[GP1:90,1] + 103.369;
   1:  PR[GP1:91,2] = PR[GP1:90,2] + 117.177;
   1:L PR[91] 10mm/sec FINE;
   1:  PR[GP1:91,1] = PR[GP1:90,1] + 101.702;
   1:  PR[GP1:91,2] = PR[GP1:90,2] + 116.916;
   1:L PR[91] 10mm/sec FINE;
   1:  PR[GP1:91,1] = PR[GP1:90,1] + 99.392;
   1:  PR[GP1:91,2] = PR[GP1:90,2] + 116.452;
   1:L PR[91] 10mm/sec FINE;
   1:  PR[GP1:91,1] = PR[GP1:90,1] + 96.985;
   1:  PR[GP1:91,2] = PR[GP1:90,2] + 115.572;
   1:L PR[91] 10mm/sec FINE;
   1:  PR[GP1:91,1] = PR[GP1:90,1] + 95.605;
   1:  PR[GP1:91,2] = PR[GP1:90,2] + 115.031;
   1:L PR[91] 10mm/sec FINE;
   1:  PR[GP1:91,1] = PR[GP1:90,1] + 95.446;
   1:  PR[GP1:91,2] = PR[GP1:90,2] + 114.948;
   1:L PR[91] 10mm/sec FINE;
   1:  PR[GP1:91,1] = PR[GP1:90,1] + 92.359;
   1:  PR[GP1:91,2] = PR[GP1:90,2] + 112.964;
   1:L PR[91] 10mm/sec FINE;
   1:  PR[GP1:91,1] = PR[GP1:90,1] + 91.932;
   1:  PR[GP1:91,2] = PR[GP1:90,2] + 112.589;
   1:L PR[91] 10mm/sec FINE;
   1:  PR[GP1:91,1] = PR[GP1:90,1] + 89.773;
   1:  PR[GP1:91,2] = PR[GP1:90,2] + 110.257;
   1:L PR[91] 10mm/sec FINE;
   1:  PR[GP1:91,1] = PR[GP1:90,1] + 89.549;
   1:  PR[GP1:91,2] = PR[GP1:90,2] + 109.980;
   1:L PR[91] 10mm/sec FINE;
   1:  PR[GP1:91,1] = PR[GP1:90,1] + 89.377;
   1:  PR[GP1:91,2] = PR[GP1:90,2] + 109.674;
   1:L PR[91] 10mm/sec FINE;
   1:  PR[GP1:91,1] = PR[GP1:90,1] + 87.862;
   1:  PR[GP1:91,2] = PR[GP1:90,2] + 106.785;
   1:L PR[91] 10mm/sec FINE;
   1:  PR[GP1:91,1] = PR[GP1:90,1] + 87.768;
   1:  PR[GP1:91,2] = PR[GP1:90,2] + 106.525;
   1:L PR[91] 10mm/sec FINE;
   1:  PR[GP1:91,1] = PR[GP1:90,1] + 87.033;
   1:  PR[GP1:91,2] = PR[GP1:90,2] + 103.354;
   1:L PR[91] 10mm/sec FINE;
   1:  PR[GP1:91,1] = PR[GP1:90,1] + 86.967;
   1:  PR[GP1:91,2] = PR[GP1:90,2] + 102.996;
   1:L PR[91] 10mm/sec FINE;
   1:  PR[GP1:91,1] = PR[GP1:90,1] + 86.960;
   1:  PR[GP1:91,2] = PR[GP1:90,2] + 102.627;
   1:L PR[91] 10mm/sec FINE;
   1:  PR[GP1:91,1] = PR[GP1:90,1] + 87.128;
   1:  PR[GP1:91,2] = PR[GP1:90,2] + 99.435;
   1:L PR[91] 10mm/sec FINE;
   1:  PR[GP1:91,1] = PR[GP1:90,1] + 87.222;
   1:  PR[GP1:91,2] = PR[GP1:90,2] + 98.861;
   1:L PR[91] 10mm/sec FINE;
   1:  PR[GP1:91,1] = PR[GP1:90,1] + 87.457;
   1:  PR[GP1:91,2] = PR[GP1:90,2] + 97.974;
   1:L PR[91] 10mm/sec FINE;
   1:  PR[GP1:91,1] = PR[GP1:90,1] + 88.815;
   1:  PR[GP1:91,2] = PR[GP1:90,2] + 94.050;
   1:L PR[91] 10mm/sec FINE;
   1:  PR[GP1:91,1] = PR[GP1:90,1] + 89.682;
   1:  PR[GP1:91,2] = PR[GP1:90,2] + 93.507;
   1:  PR[GP1:91,3] = PR[GP1:90,3] + 63.900;
   1:L PR[91] 10mm/sec FINE;
   1:  PR[GP1:91,1] = PR[GP1:90,1] + 91.688;
   1:  PR[GP1:91,2] = PR[GP1:90,2] + 90.143;
   1:L PR[91] 10mm/sec FINE;
   1:  PR[GP1:91,1] = PR[GP1:90,1] + 93.014;
   1:  PR[GP1:91,2] = PR[GP1:90,2] + 88.305;
   1:L PR[91] 10mm/sec FINE;
   1:  PR[GP1:91,1] = PR[GP1:90,1] + 95.211;
   1:  PR[GP1:91,2] = PR[GP1:90,2] + 85.925;
   1:L PR[91] 10mm/sec FINE;
   1:  PR[GP1:91,1] = PR[GP1:90,1] + 95.988;
   1:  PR[GP1:91,2] = PR[GP1:90,2] + 85.121;
   1:L PR[91] 10mm/sec FINE;
   1:  PR[GP1:91,1] = PR[GP1:90,1] + 99.047;
   1:  PR[GP1:91,2] = PR[GP1:90,2] + 82.728;
   1:L PR[91] 10mm/sec FINE;
   1:  PR[GP1:91,1] = PR[GP1:90,1] + 100.377;
   1:  PR[GP1:91,2] = PR[GP1:90,2] + 81.740;
   1:L PR[91] 10mm/sec FINE;
   1:  PR[GP1:91,1] = PR[GP1:90,1] + 104.078;
   1:  PR[GP1:91,2] = PR[GP1:90,2] + 79.747;
   1:L PR[91] 10mm/sec FINE;
   1:  PR[GP1:91,1] = PR[GP1:90,1] + 105.301;
   1:  PR[GP1:91,2] = PR[GP1:90,2] + 79.030;
   1:L PR[91] 10mm/sec FINE;
   1:  PR[GP1:91,1] = PR[GP1:90,1] + 111.458;
   1:  PR[GP1:91,2] = PR[GP1:90,2] + 76.687;
   1:L PR[91] 10mm/sec FINE;
   1:  PR[GP1:91,1] = PR[GP1:90,1] + 116.273;
   1:  PR[GP1:91,2] = PR[GP1:90,2] + 75.735;
   1:L PR[91] 10mm/sec FINE;
   1:  PR[GP1:91,1] = PR[GP1:90,1] + 119.300;
   1:  PR[GP1:91,2] = PR[GP1:90,2] + 75.560;
   1:L PR[91] 10mm/sec FINE;
   1:  PR[GP1:91,1] = PR[GP1:90,1] + 120.237;
   1:  PR[GP1:91,2] = PR[GP1:90,2] + 75.550;
   1:L PR[91] 10mm/sec FINE;
   1:  PR[GP1:91,1] = PR[GP1:90,1] + 123.586;
   1:  PR[GP1:91,2] = PR[GP1:90,2] + 75.828;
   1:L PR[91] 10mm/sec FINE;
   1:  PR[GP1:91,1] = PR[GP1:90,1] + 126.502;
   1:  PR[GP1:91,2] = PR[GP1:90,2] + 76.603;
   1:L PR[91] 10mm/sec FINE;
   1:  PR[GP1:91,1] = PR[GP1:90,1] + 127.478;
   1:  PR[GP1:91,2] = PR[GP1:90,2] + 76.980;
   1:L PR[91] 10mm/sec FINE;
   1:  PR[GP1:91,1] = PR[GP1:90,1] + 129.884;
   1:  PR[GP1:91,2] = PR[GP1:90,2] + 78.090;
   1:L PR[91] 10mm/sec FINE;
   1:  PR[GP1:91,1] = PR[GP1:90,1] + 131.521;
   1:  PR[GP1:91,2] = PR[GP1:90,2] + 79.256;
   1:L PR[91] 10mm/sec FINE;
   1:  PR[GP1:91,1] = PR[GP1:90,1] + 132.919;
   1:  PR[GP1:91,2] = PR[GP1:90,2] + 80.355;
   1:L PR[91] 10mm/sec FINE;
   1:  PR[GP1:91,1] = PR[GP1:90,1] + 134.224;
   1:  PR[GP1:91,2] = PR[GP1:90,2] + 81.747;
   1:L PR[91] 10mm/sec FINE;
   1:  PR[GP1:91,1] = PR[GP1:90,1] + 135.175;
   1:  PR[GP1:91,2] = PR[GP1:90,2] + 83.164;
   1:L PR[91] 10mm/sec FINE;
   1:  PR[GP1:91,1] = PR[GP1:90,1] + 136.125;
   1:  PR[GP1:91,2] = PR[GP1:90,2] + 84.742;
   1:L PR[91] 10mm/sec FINE;
   1:  PR[GP1:91,1] = PR[GP1:90,1] + 136.748;
   1:  PR[GP1:91,2] = PR[GP1:90,2] + 86.555;
   1:L PR[91] 10mm/sec FINE;
   1:  PR[GP1:91,1] = PR[GP1:90,1] + 137.151;
   1:  PR[GP1:91,2] = PR[GP1:90,2] + 87.795;
   1:L PR[91] 10mm/sec FINE;
   1:  PR[GP1:91,1] = PR[GP1:90,1] + 137.417;
   1:  PR[GP1:91,2] = PR[GP1:90,2] + 89.881;
   1:L PR[91] 10mm/sec FINE;
   1:  PR[GP1:91,1] = PR[GP1:90,1] + 137.511;
   1:  PR[GP1:91,2] = PR[GP1:90,2] + 90.860;
   1:L PR[91] 10mm/sec FINE;
   1:  PR[GP1:91,1] = PR[GP1:90,1] + 137.354;
   1:  PR[GP1:91,2] = PR[GP1:90,2] + 93.337;
   1:L PR[91] 10mm/sec FINE;
   1:  PR[GP1:91,1] = PR[GP1:90,1] + 137.296;
   1:  PR[GP1:91,2] = PR[GP1:90,2] + 94.021;
   1:L PR[91] 10mm/sec FINE;
   1:  PR[GP1:91,1] = PR[GP1:90,1] + 136.512;
   1:  PR[GP1:91,2] = PR[GP1:90,2] + 97.278;
   1:L PR[91] 10mm/sec FINE;
   1:  PR[GP1:91,1] = PR[GP1:90,1] + 136.226;
   1:  PR[GP1:91,2] = PR[GP1:90,2] + 98.000;
   1:L PR[91] 10mm/sec FINE;
   1:  PR[GP1:91,1] = PR[GP1:90,1] + 135.316;
   1:  PR[GP1:91,2] = PR[GP1:90,2] + 100.026;
   1:L PR[91] 10mm/sec FINE;
   1:  PR[GP1:91,1] = PR[GP1:90,1] + 133.851;
   1:  PR[GP1:91,2] = PR[GP1:90,2] + 102.482;
   1:L PR[91] 10mm/sec FINE;
   1:  PR[GP1:91,1] = PR[GP1:90,1] + 133.482;
   1:  PR[GP1:91,2] = PR[GP1:90,2] + 103.002;
   1:L PR[91] 10mm/sec FINE;
   1:  PR[GP1:91,1] = PR[GP1:90,1] + 132.253;
   1:  PR[GP1:91,2] = PR[GP1:90,2] + 104.629;
   1:L PR[91] 10mm/sec FINE;
   1:  PR[GP1:91,1] = PR[GP1:90,1] + 131.549;
   1:  PR[GP1:91,2] = PR[GP1:90,2] + 105.470;
   1:L PR[91] 10mm/sec FINE;
   1:  PR[GP1:91,1] = PR[GP1:90,1] + 130.529;
   1:  PR[GP1:91,2] = PR[GP1:90,2] + 106.564;
   1:L PR[91] 10mm/sec FINE;
   1:  PR[GP1:91,1] = PR[GP1:90,1] + 129.364;
   1:  PR[GP1:91,2] = PR[GP1:90,2] + 107.739;
   1:L PR[91] 10mm/sec FINE;
   1:  PR[GP1:91,1] = PR[GP1:90,1] + 127.972;
   1:  PR[GP1:91,2] = PR[GP1:90,2] + 108.976;
   1:L PR[91] 10mm/sec FINE;
   1:  PR[GP1:91,1] = PR[GP1:90,1] + 124.743;
   1:  PR[GP1:91,2] = PR[GP1:90,2] + 111.371;
   1:L PR[91] 10mm/sec FINE;
   1:  PR[GP1:91,1] = PR[GP1:90,1] + 124.724;
   1:  PR[GP1:91,2] = PR[GP1:90,2] + 111.400;
   1:L PR[91] 10mm/sec FINE;
   1:  PR[GP1:91,1] = PR[GP1:90,1] + 124.231;
   1:  PR[GP1:91,2] = PR[GP1:90,2] + 111.734;
   1:L PR[91] 10mm/sec FINE;
   1:  PR[GP1:91,1] = PR[GP1:90,1] + 124.029;
   1:  PR[GP1:91,2] = PR[GP1:90,2] + 111.850;
   1:L PR[91] 10mm/sec FINE;
   1:  PR[GP1:91,1] = PR[GP1:90,1] + 123.620;
   1:  PR[GP1:91,2] = PR[GP1:90,2] + 112.141;
   1:L PR[91] 10mm/sec FINE;
   1:  PR[GP1:91,1] = PR[GP1:90,1] + 122.920;
   1:  PR[GP1:91,2] = PR[GP1:90,2] + 112.528;
   1:L PR[91] 10mm/sec FINE;
   1:  PR[GP1:91,1] = PR[GP1:90,1] + 122.771;
   1:  PR[GP1:91,2] = PR[GP1:90,2] + 112.595;
   1:L PR[91] 10mm/sec FINE;
   1:  PR[GP1:91,1] = PR[GP1:90,1] + 121.414;
   1:  PR[GP1:91,2] = PR[GP1:90,2] + 113.522;
   1:L PR[91] 10mm/sec FINE;
   1:  PR[GP1:91,1] = PR[GP1:90,1] + 121.126;
   1:  PR[GP1:91,2] = PR[GP1:90,2] + 113.664;
   1:L PR[91] 10mm/sec FINE;
   1:  PR[GP1:91,1] = PR[GP1:90,1] + 120.953;
   1:  PR[GP1:91,2] = PR[GP1:90,2] + 113.726;
   1:L PR[91] 10mm/sec FINE;
   1:  PR[GP1:91,1] = PR[GP1:90,1] + 118.830;
   1:  PR[GP1:91,2] = PR[GP1:90,2] + 114.735;
   1:L PR[91] 10mm/sec FINE;
   1:  PR[GP1:91,1] = PR[GP1:90,1] + 117.653;
   1:  PR[GP1:91,2] = PR[GP1:90,2] + 115.323;
   1:L PR[91] 10mm/sec FINE;
   1:  PR[GP1:91,1] = PR[GP1:90,1] + 116.355;
   1:  PR[GP1:91,2] = PR[GP1:90,2] + 115.704;
   1:L PR[91] 10mm/sec FINE;
   1:  PR[GP1:91,1] = PR[GP1:90,1] + 113.771;
   1:  PR[GP1:91,2] = PR[GP1:90,2] + 116.506;
   1:L PR[91] 10mm/sec FINE;
   1:  PR[GP1:91,1] = PR[GP1:90,1] + 109.868;
   1:  PR[GP1:91,2] = PR[GP1:90,2] + 117.011;
   1:L PR[91] 10mm/sec FINE;
   1:  PR[GP1:91,1] = PR[GP1:90,1] + 107.916;
   1:  PR[GP1:91,2] = PR[GP1:90,2] + 117.008;
   1:L PR[91] 10mm/sec FINE;
   1:  PR[GP1:91,1] = PR[GP1:90,1] + 104.026;
   1:  PR[GP1:91,2] = PR[GP1:90,2] + 116.855;
   1:L PR[91] 10mm/sec FINE;
   1:  PR[GP1:91,1] = PR[GP1:90,1] + 102.911;
   1:  PR[GP1:91,2] = PR[GP1:90,2] + 116.681;
   1:L PR[91] 10mm/sec FINE;
   1:  PR[GP1:91,1] = PR[GP1:90,1] + 100.108;
   1:  PR[GP1:91,2] = PR[GP1:90,2] + 116.118;
   1:L PR[91] 10mm/sec FINE;
   1:  PR[GP1:91,1] = PR[GP1:90,1] + 98.213;
   1:  PR[GP1:91,2] = PR[GP1:90,2] + 115.425;
   1:L PR[91] 10mm/sec FINE;
   1:  PR[GP1:91,1] = PR[GP1:90,1] + 96.377;
   1:  PR[GP1:91,2] = PR[GP1:90,2] + 114.705;
   1:L PR[91] 10mm/sec FINE;
   1:  PR[GP1:91,1] = PR[GP1:90,1] + 96.160;
   1:  PR[GP1:91,2] = PR[GP1:90,2] + 114.592;
   1:L PR[91] 10mm/sec FINE;
   1:  PR[GP1:91,1] = PR[GP1:90,1] + 93.225;
   1:  PR[GP1:91,2] = PR[GP1:90,2] + 112.708;
   1:L PR[91] 10mm/sec FINE;
   1:  PR[GP1:91,1] = PR[GP1:90,1] + 92.553;
   1:  PR[GP1:91,2] = PR[GP1:90,2] + 112.117;
   1:L PR[91] 10mm/sec FINE;
   1:  PR[GP1:91,1] = PR[GP1:90,1] + 90.750;
   1:  PR[GP1:91,2] = PR[GP1:90,2] + 110.169;
   1:L PR[91] 10mm/sec FINE;
   1:  PR[GP1:91,1] = PR[GP1:90,1] + 90.305;
   1:  PR[GP1:91,2] = PR[GP1:90,2] + 109.620;
   1:L PR[91] 10mm/sec FINE;
   1:  PR[GP1:91,1] = PR[GP1:90,1] + 89.965;
   1:  PR[GP1:91,2] = PR[GP1:90,2] + 109.014;
   1:L PR[91] 10mm/sec FINE;
   1:  PR[GP1:91,1] = PR[GP1:90,1] + 88.699;
   1:  PR[GP1:91,2] = PR[GP1:90,2] + 106.600;
   1:L PR[91] 10mm/sec FINE;
   1:  PR[GP1:91,1] = PR[GP1:90,1] + 88.489;
   1:  PR[GP1:91,2] = PR[GP1:90,2] + 106.013;
   1:L PR[91] 10mm/sec FINE;
   1:  PR[GP1:91,1] = PR[GP1:90,1] + 87.874;
   1:  PR[GP1:91,2] = PR[GP1:90,2] + 103.364;
   1:L PR[91] 10mm/sec FINE;
   1:  PR[GP1:91,1] = PR[GP1:90,1] + 87.748;
   1:  PR[GP1:91,2] = PR[GP1:90,2] + 102.677;
   1:L PR[91] 10mm/sec FINE;
   1:  PR[GP1:91,1] = PR[GP1:90,1] + 87.734;
   1:  PR[GP1:91,2] = PR[GP1:90,2] + 101.969;
   1:L PR[91] 10mm/sec FINE;
   1:  PR[GP1:91,1] = PR[GP1:90,1] + 87.875;
   1:  PR[GP1:91,2] = PR[GP1:90,2] + 99.303;
   1:L PR[91] 10mm/sec FINE;
   1:  PR[GP1:91,1] = PR[GP1:90,1] + 88.015;
   1:  PR[GP1:91,2] = PR[GP1:90,2] + 98.436;
   1:L PR[91] 10mm/sec FINE;
   1:  PR[GP1:91,1] = PR[GP1:90,1] + 88.139;
   1:  PR[GP1:91,2] = PR[GP1:90,2] + 97.968;
   1:L PR[91] 10mm/sec FINE;
   1:  PR[GP1:91,1] = PR[GP1:90,1] + 89.125;
   1:  PR[GP1:91,2] = PR[GP1:90,2] + 95.121;
   1:L PR[91] 10mm/sec FINE;
   1:  PR[GP1:91,1] = PR[GP1:90,1] + 89.563;
   1:  PR[GP1:91,2] = PR[GP1:90,2] + 93.763;
   1:L PR[91] 10mm/sec FINE;
   1:  PR[GP1:91,1] = PR[GP1:90,1] + 90.601;
   1:  PR[GP1:91,2] = PR[GP1:90,2] + 92.828;
   1:  PR[GP1:91,3] = PR[GP1:90,3] + 64.900;
   1:L PR[91] 10mm/sec FINE;
   1:  PR[GP1:91,1] = PR[GP1:90,1] + 92.212;
   1:  PR[GP1:91,2] = PR[GP1:90,2] + 90.127;
   1:L PR[91] 10mm/sec FINE;
   1:  PR[GP1:91,1] = PR[GP1:90,1] + 94.027;
   1:  PR[GP1:91,2] = PR[GP1:90,2] + 87.612;
   1:L PR[91] 10mm/sec FINE;
   1:  PR[GP1:91,1] = PR[GP1:90,1] + 95.791;
   1:  PR[GP1:91,2] = PR[GP1:90,2] + 85.700;
   1:L PR[91] 10mm/sec FINE;
   1:  PR[GP1:91,1] = PR[GP1:90,1] + 96.714;
   1:  PR[GP1:91,2] = PR[GP1:90,2] + 84.745;
   1:L PR[91] 10mm/sec FINE;
   1:  PR[GP1:91,1] = PR[GP1:90,1] + 100.344;
   1:  PR[GP1:91,2] = PR[GP1:90,2] + 81.906;
   1:L PR[91] 10mm/sec FINE;
   1:  PR[GP1:91,1] = PR[GP1:90,1] + 101.080;
   1:  PR[GP1:91,2] = PR[GP1:90,2] + 81.359;
   1:L PR[91] 10mm/sec FINE;
   1:  PR[GP1:91,1] = PR[GP1:90,1] + 103.140;
   1:  PR[GP1:91,2] = PR[GP1:90,2] + 80.250;
   1:L PR[91] 10mm/sec FINE;
   1:  PR[GP1:91,1] = PR[GP1:90,1] + 106.081;
   1:  PR[GP1:91,2] = PR[GP1:90,2] + 78.527;
   1:L PR[91] 10mm/sec FINE;
   1:  PR[GP1:91,1] = PR[GP1:90,1] + 112.440;
   1:  PR[GP1:91,2] = PR[GP1:90,2] + 76.102;
   1:L PR[91] 10mm/sec FINE;
   1:  PR[GP1:91,1] = PR[GP1:90,1] + 117.064;
   1:  PR[GP1:91,2] = PR[GP1:90,2] + 75.192;
   1:L PR[91] 10mm/sec FINE;
   1:  PR[GP1:91,1] = PR[GP1:90,1] + 120.572;
   1:  PR[GP1:91,2] = PR[GP1:90,2] + 74.990;
   1:L PR[91] 10mm/sec FINE;
   1:  PR[GP1:91,1] = PR[GP1:90,1] + 120.885;
   1:  PR[GP1:91,2] = PR[GP1:90,2] + 74.987;
   1:L PR[91] 10mm/sec FINE;
   1:  PR[GP1:91,1] = PR[GP1:90,1] + 122.056;
   1:  PR[GP1:91,2] = PR[GP1:90,2] + 75.084;
   1:L PR[91] 10mm/sec FINE;
   1:  PR[GP1:91,1] = PR[GP1:90,1] + 123.470;
   1:  PR[GP1:91,2] = PR[GP1:90,2] + 75.267;
   1:L PR[91] 10mm/sec FINE;
   1:  PR[GP1:91,1] = PR[GP1:90,1] + 124.631;
   1:  PR[GP1:91,2] = PR[GP1:90,2] + 75.394;
   1:L PR[91] 10mm/sec FINE;
   1:  PR[GP1:91,1] = PR[GP1:90,1] + 126.981;
   1:  PR[GP1:91,2] = PR[GP1:90,2] + 76.020;
   1:L PR[91] 10mm/sec FINE;
   1:  PR[GP1:91,1] = PR[GP1:90,1] + 128.773;
   1:  PR[GP1:91,2] = PR[GP1:90,2] + 76.712;
   1:L PR[91] 10mm/sec FINE;
   1:  PR[GP1:91,1] = PR[GP1:90,1] + 130.703;
   1:  PR[GP1:91,2] = PR[GP1:90,2] + 77.603;
   1:L PR[91] 10mm/sec FINE;
   1:  PR[GP1:91,1] = PR[GP1:90,1] + 132.015;
   1:  PR[GP1:91,2] = PR[GP1:90,2] + 78.538;
   1:L PR[91] 10mm/sec FINE;
   1:  PR[GP1:91,1] = PR[GP1:90,1] + 133.908;
   1:  PR[GP1:91,2] = PR[GP1:90,2] + 80.025;
   1:L PR[91] 10mm/sec FINE;
   1:  PR[GP1:91,1] = PR[GP1:90,1] + 134.953;
   1:  PR[GP1:91,2] = PR[GP1:90,2] + 81.140;
   1:L PR[91] 10mm/sec FINE;
   1:  PR[GP1:91,1] = PR[GP1:90,1] + 136.202;
   1:  PR[GP1:91,2] = PR[GP1:90,2] + 83.002;
   1:L PR[91] 10mm/sec FINE;
   1:  PR[GP1:91,1] = PR[GP1:90,1] + 136.963;
   1:  PR[GP1:91,2] = PR[GP1:90,2] + 84.267;
   1:L PR[91] 10mm/sec FINE;
   1:  PR[GP1:91,1] = PR[GP1:90,1] + 137.463;
   1:  PR[GP1:91,2] = PR[GP1:90,2] + 85.719;
   1:L PR[91] 10mm/sec FINE;
   1:  PR[GP1:91,1] = PR[GP1:90,1] + 138.003;
   1:  PR[GP1:91,2] = PR[GP1:90,2] + 87.382;
   1:L PR[91] 10mm/sec FINE;
   1:  PR[GP1:91,1] = PR[GP1:90,1] + 138.217;
   1:  PR[GP1:91,2] = PR[GP1:90,2] + 89.056;
   1:L PR[91] 10mm/sec FINE;
   1:  PR[GP1:91,1] = PR[GP1:90,1] + 138.351;
   1:  PR[GP1:91,2] = PR[GP1:90,2] + 90.452;
   1:L PR[91] 10mm/sec FINE;
   1:  PR[GP1:91,1] = PR[GP1:90,1] + 138.225;
   1:  PR[GP1:91,2] = PR[GP1:90,2] + 92.440;
   1:L PR[91] 10mm/sec FINE;
   1:  PR[GP1:91,1] = PR[GP1:90,1] + 138.127;
   1:  PR[GP1:91,2] = PR[GP1:90,2] + 93.596;
   1:L PR[91] 10mm/sec FINE;
   1:  PR[GP1:91,1] = PR[GP1:90,1] + 137.351;
   1:  PR[GP1:91,2] = PR[GP1:90,2] + 96.803;
   1:L PR[91] 10mm/sec FINE;
   1:  PR[GP1:91,1] = PR[GP1:90,1] + 136.273;
   1:  PR[GP1:91,2] = PR[GP1:90,2] + 99.525;
   1:L PR[91] 10mm/sec FINE;
   1:  PR[GP1:91,1] = PR[GP1:90,1] + 136.101;
   1:  PR[GP1:91,2] = PR[GP1:90,2] + 99.843;
   1:L PR[91] 10mm/sec FINE;
   1:  PR[GP1:91,1] = PR[GP1:90,1] + 134.759;
   1:  PR[GP1:91,2] = PR[GP1:90,2] + 102.092;
   1:L PR[91] 10mm/sec FINE;
